LIN {X 0,Y 516.944,Z 452.093,A -85,B 0,C 180,E1 -4929.732,E2 -4929.732} C_VEL
LIN {X 0,Y 516.912,Z 452.096,A -85,B 0,C 180,E1 -4932.596,E2 -4932.596} C_VEL
LIN {X 0,Y 516.948,Z 452.092,A -85,B 0,C 180,E1 -4935.03,E2 -4935.03} C_VEL
LIN {X 0,Y 516.971,Z 452.089,A -85,B 0,C 180,E1 -4938.234,E2 -4938.234} C_VEL
LIN {X 0,Y 516.971,Z 452.089,A -85,B 0,C 180,E1 -4941.4,E2 -4941.4} C_VEL
LIN {X 0,Y 517.028,Z 452.081,A -85,B 0,C 180,E1 -4944.54,E2 -4944.54} C_VEL
LIN {X 0,Y 517.089,Z 452.074,A -85,B 0,C 180,E1 -4947.663,E2 -4947.663} C_VEL
LIN {X 0,Y 517.097,Z 452.071,A -85,B 0,C 180,E1 -4950.779,E2 -4950.779} C_VEL
LIN {X 0,Y 517.016,Z 452.085,A -85,B 0,C 180,E1 -4953.117,E2 -4953.117} C_VEL
LIN {X 0,Y 517.016,Z 452.085,A -85,B 0,C 180,E1 -4956.243,E2 -4956.243} C_VEL
LIN {X 0,Y 516.954,Z 452.092,A -85,B 0,C 180,E1 -4959.389,E2 -4959.389} C_VEL
LIN {X 0,Y 516.958,Z 452.09,A -85,B 0,C 180,E1 -4961.807,E2 -4961.807} C_VEL
LIN {X 0,Y 516.95,Z 452.09,A -85,B 0,C 180,E1 -4965.147,E2 -4965.147} C_VEL
LIN {X 0,Y 516.93,Z 452.093,A -85,B 0,C 180,E1 -4968.222,E2 -4968.222} C_VEL
LIN {X 0,Y 516.918,Z 452.097,A -85,B 0,C 180,E1 -4970.701,E2 -4970.701} C_VEL
LIN {X 0,Y 516.909,Z 452.097,A -85,B 0,C 180,E1 -4974.072,E2 -4974.072} C_VEL
LIN {X 0,Y 516.93,Z 452.097,A -85,B 0,C 180,E1 -4976.658,E2 -4976.658} C_VEL
LIN {X 0,Y 516.916,Z 452.096,A -85,B 0,C 180,E1 -4979.524,E2 -4979.524} C_VEL
LIN {X 0,Y 516.9,Z 452.098,A -85,B 0,C 180,E1 -4982.543,E2 -4982.543} C_VEL
LIN {X 0,Y 516.871,Z 452.1,A -85,B 0,C 180,E1 -4985.33,E2 -4985.33} C_VEL
LIN {X 0,Y 516.885,Z 452.101,A -85,B 0,C 180,E1 -4987.943,E2 -4987.943} C_VEL
LIN {X 0,Y 516.889,Z 452.101,A -85,B 0,C 180,E1 -4990.741,E2 -4990.741} C_VEL
LIN {X 0,Y 516.887,Z 452.099,A -85,B 0,C 180,E1 -4992.831,E2 -4992.831} C_VEL
LIN {X 0,Y 516.887,Z 452.099,A -85,B 0,C 180,E1 -4996.097,E2 -4996.097} C_VEL
LIN {X 0,Y 516.92,Z 452.098,A -85,B 0,C 180,E1 -4998.398,E2 -4998.398} C_VEL
LIN {X 0,Y 516.884,Z 452.099,A -85,B 0,C 180,E1 -5001.284,E2 -5001.284} C_VEL
LIN {X 0,Y 516.808,Z 452.109,A -85,B 0,C 180,E1 -5004.214,E2 -5004.214} C_VEL
LIN {X 0,Y 516.707,Z 452.125,A -85,B 0,C 180,E1 -5006.105,E2 -5006.105} C_VEL
LIN {X 0,Y 516.479,Z 452.226,A -85,B 0,C 180,E1 -5007.947,E2 -5007.947} C_VEL
LIN {X 0,Y 516.445,Z 455.171,A -85,B 0,C 180,E1 -5010.665,E2 -5010.665} C_VEL
LIN {X 0,Y 516.432,Z 458.051,A -85,B 0,C 180,E1 -5013.314,E2 -5013.314} C_VEL
LIN {X 0,Y 516.375,Z 460.913,A -85,B 0,C 180,E1 -5015.901,E2 -5015.901} C_VEL
LIN {X 0,Y 516.337,Z 463.731,A -85,B 0,C 180,E1 -5018.438,E2 -5018.438} C_VEL
LIN {X 0,Y 516.302,Z 466.547,A -85,B 0,C 180,E1 -5020.932,E2 -5020.932} C_VEL
LIN {X 0,Y 516.277,Z 469.313,A -85,B 0,C 180,E1 -5023.389,E2 -5023.389} C_VEL
LIN {X 0,Y 516.308,Z 472.56,A -85,B 0,C 180,E1 -5026.219,E2 -5026.219} C_VEL
LIN {X 0,Y 518.389,Z 484.619,A -85,B 0,C 180,E1 -5026.6,E2 -5026.6} C_VEL
LIN {X 0,Y 518.151,Z 497.874,A -85,B 0,C 180,E1 -5027.117,E2 -5027.117} C_VEL
LIN {X 0,Y 517.878,Z 509.167,A -85,B 0,C 180,E1 -5027.715,E2 -5027.715} C_VEL
LIN {X 0,Y 517.621,Z 519.986,A -85,B 0,C 180,E1 -5028.447,E2 -5028.447} C_VEL
LIN {X 0,Y 517.303,Z 530.501,A -85,B 0,C 180,E1 -5029.332,E2 -5029.332} C_VEL
LIN {X 0,Y 517.054,Z 539.091,A -85,B 0,C 180,E1 -5030.218,E2 -5030.218} C_VEL
LIN {X 0,Y 516.835,Z 546.997,A -85,B 0,C 180,E1 -5031.2,E2 -5031.2} C_VEL
LIN {X 0,Y 516.602,Z 554.73,A -85,B 0,C 180,E1 -5032.378,E2 -5032.378} C_VEL
LIN {X 0,Y 516.448,Z 561.797,A -85,B 0,C 180,E1 -5033.75,E2 -5033.75} C_VEL
LIN {X 0,Y 516.314,Z 566.51,A -85,B 0,C 180,E1 -5034.924,E2 -5034.924} C_VEL
LIN {X 0,Y 516.373,Z 570.109,A -85,B 0,C 180,E1 -5036.098,E2 -5036.098} C_VEL
LIN {X 0,Y 516.283,Z 571.978,A -85,B 0,C 180,E1 -5036.879,E2 -5036.879} C_VEL
LIN {X 0,Y 516.261,Z 573.384,A -85,B 0,C 180,E1 -5037.659,E2 -5037.659} C_VEL
LIN {X 0,Y 516.161,Z 575.003,A -85,B 0,C 180,E1 -5039.22,E2 -5039.22} C_VEL
LIN {X 0,Y 516.154,Z 575.245,A -85,B 0,C 180,E1 -5040,E2 -5040} C_VEL
LIN {X 0,Y 516.16,Z 575.064,A -85,B 0,C 180,E1 -5040.78,E2 -5040.78} C_VEL
LIN {X 0,Y 516.261,Z 573.525,A -85,B 0,C 180,E1 -5042.34,E2 -5042.34} C_VEL
LIN {X 0,Y 516.283,Z 572.181,A -85,B 0,C 180,E1 -5043.121,E2 -5043.121} C_VEL
LIN {X 0,Y 516.361,Z 569.332,A -85,B 0,C 180,E1 -5044.293,E2 -5044.293} C_VEL
LIN {X 0,Y 516.401,Z 565.469,A -85,B 0,C 180,E1 -5045.467,E2 -5045.467} C_VEL
LIN {X 0,Y 516.49,Z 559.63,A -85,B 0,C 180,E1 -5046.814,E2 -5046.814} C_VEL
LIN {X 0,Y 516.653,Z 552.961,A -85,B 0,C 180,E1 -5048.015,E2 -5048.015} C_VEL
LIN {X 0,Y 516.849,Z 544.818,A -85,B 0,C 180,E1 -5049.194,E2 -5049.194} C_VEL
LIN {X 0,Y 517.107,Z 536.463,A -85,B 0,C 180,E1 -5050.177,E2 -5050.177} C_VEL
LIN {X 0,Y 517.465,Z 526.118,A -85,B 0,C 180,E1 -5051.159,E2 -5051.159} C_VEL
LIN {X 0,Y 517.787,Z 514.576,A -85,B 0,C 180,E1 -5052.037,E2 -5052.037} C_VEL
LIN {X 0,Y 518.071,Z 502.798,A -85,B 0,C 180,E1 -5052.735,E2 -5052.735} C_VEL
LIN {X 0,Y 518.336,Z 490.688,A -85,B 0,C 180,E1 -5053.277,E2 -5053.277} C_VEL
LIN {X 0,Y 518.251,Z 483.303,A -85,B 0,C 180,E1 -5053.541,E2 -5053.541} C_VEL
LIN {X 0,Y 516.316,Z 472.997,A -85,B 0,C 180,E1 -5053.881,E2 -5053.881} C_VEL
LIN {X 0,Y 516.34,Z 470.114,A -85,B 0,C 180,E1 -5056.609,E2 -5056.609} C_VEL
LIN {X 0,Y 516.386,Z 467.623,A -85,B 0,C 180,E1 -5059.065,E2 -5059.065} C_VEL
LIN {X 0,Y 516.433,Z 465.115,A -85,B 0,C 180,E1 -5061.558,E2 -5061.558} C_VEL
LIN {X 0,Y 516.557,Z 462.467,A -85,B 0,C 180,E1 -5064.277,E2 -5064.277} C_VEL
LIN {X 0,Y 516.677,Z 459.367,A -85,B 0,C 180,E1 -5067.547,E2 -5067.547} C_VEL
LIN {X 0,Y 516.708,Z 456.952,A -85,B 0,C 180,E1 -5070.216,E2 -5070.216} C_VEL
LIN {X 0,Y 516.837,Z 454.601,A -85,B 0,C 180,E1 -5072.951,E2 -5072.951} C_VEL
LIN {X 0,Y 516.847,Z 452.379,A -85,B 0,C 180,E1 -5075.782,E2 -5075.782} C_VEL
LIN {X 0,Y 516.883,Z 452.104,A -85,B 0,C 180,E1 -5077.943,E2 -5077.943} C_VEL
LIN {X 0,Y 516.887,Z 452.102,A -85,B 0,C 180,E1 -5080.741,E2 -5080.741} C_VEL
LIN {X 0,Y 516.908,Z 452.1,A -85,B 0,C 180,E1 -5082.829,E2 -5082.829} C_VEL
LIN {X 0,Y 516.926,Z 452.098,A -85,B 0,C 180,E1 -5085.01,E2 -5085.01} C_VEL
LIN {X 0,Y 516.918,Z 452.098,A -85,B 0,C 180,E1 -5088.398,E2 -5088.398} C_VEL
LIN {X 0,Y 516.932,Z 452.198,A -85,B 0,C 180,E1 -5089.263,E2 -5089.263} C_VEL
LIN {X 0,Y 517.422,Z 454.988,A -85,B 0,C 180,E1 -5091.332,E2 -5091.332} C_VEL
LIN {X 0,Y 518.009,Z 458.473,A -85,B 0,C 180,E1 -5093.347,E2 -5093.347} C_VEL
LIN {X 0,Y 518.115,Z 462.532,A -85,B 0,C 180,E1 -5095.27,E2 -5095.27} C_VEL
LIN {X 0,Y 517.661,Z 469.386,A -85,B 0,C 180,E1 -5098.029,E2 -5098.029} C_VEL
LIN {X 0,Y 517.314,Z 476.785,A -85,B 0,C 180,E1 -5100.72,E2 -5100.72} C_VEL
LIN {X 0,Y 517.151,Z 484.588,A -85,B 0,C 180,E1 -5103.355,E2 -5103.355} C_VEL
LIN {X 0,Y 517.002,Z 492.652,A -85,B 0,C 180,E1 -5105.932,E2 -5105.932} C_VEL
LIN {X 0,Y 516.828,Z 502.252,A -85,B 0,C 180,E1 -5108.878,E2 -5108.878} C_VEL
LIN {X 0,Y 516.716,Z 511.979,A -85,B 0,C 180,E1 -5111.77,E2 -5111.77} C_VEL
LIN {X 0,Y 516.633,Z 523.068,A -85,B 0,C 180,E1 -5115.021,E2 -5115.021} C_VEL
LIN {X 0,Y 516.569,Z 526.747,A -85,B 0,C 180,E1 -5116.101,E2 -5116.101} C_VEL
LIN {X 0,Y 518.446,Z 539.825,A -85,B 0,C 180,E1 -5116.452,E2 -5116.452} C_VEL
LIN {X 0,Y 518.221,Z 551.89,A -85,B 0,C 180,E1 -5116.87,E2 -5116.87} C_VEL
LIN {X 0,Y 517.963,Z 564.239,A -85,B 0,C 180,E1 -5117.461,E2 -5117.461} C_VEL
LIN {X 0,Y 517.647,Z 575.446,A -85,B 0,C 180,E1 -5118.154,E2 -5118.154} C_VEL
LIN {X 0,Y 517.345,Z 586.795,A -85,B 0,C 180,E1 -5119.036,E2 -5119.036} C_VEL
LIN {X 0,Y 517.018,Z 596.875,A -85,B 0,C 180,E1 -5120.019,E2 -5120.019} C_VEL
LIN {X 0,Y 516.77,Z 606.653,A -85,B 0,C 180,E1 -5121.199,E2 -5121.199} C_VEL
LIN {X 0,Y 516.563,Z 614.431,A -85,B 0,C 180,E1 -5122.377,E2 -5122.377} C_VEL
LIN {X 0,Y 516.427,Z 621.594,A -85,B 0,C 180,E1 -5123.75,E2 -5123.75} C_VEL
LIN {X 0,Y 516.314,Z 626.349,A -85,B 0,C 180,E1 -5124.924,E2 -5124.924} C_VEL
LIN {X 0,Y 516.354,Z 629.957,A -85,B 0,C 180,E1 -5126.098,E2 -5126.098} C_VEL
LIN {X 0,Y 516.282,Z 631.806,A -85,B 0,C 180,E1 -5126.879,E2 -5126.879} C_VEL
LIN {X 0,Y 516.261,Z 633.192,A -85,B 0,C 180,E1 -5127.659,E2 -5127.659} C_VEL
LIN {X 0,Y 516.16,Z 634.785,A -85,B 0,C 180,E1 -5129.22,E2 -5129.22} C_VEL
LIN {X 0,Y 516.154,Z 635,A -85,B 0,C 180,E1 -5130,E2 -5130} C_VEL
LIN {X 0,Y 516.192,Z 634.183,A -85,B 0,C 180,E1 -5131.56,E2 -5131.56} C_VEL
LIN {X 0,Y 516.26,Z 633.195,A -85,B 0,C 180,E1 -5132.341,E2 -5132.341} C_VEL
LIN {X 0,Y 516.282,Z 631.81,A -85,B 0,C 180,E1 -5133.121,E2 -5133.121} C_VEL
LIN {X 0,Y 516.343,Z 628.891,A -85,B 0,C 180,E1 -5134.293,E2 -5134.293} C_VEL
LIN {X 0,Y 516.405,Z 624.912,A -85,B 0,C 180,E1 -5135.467,E2 -5135.467} C_VEL
LIN {X 0,Y 516.479,Z 618.972,A -85,B 0,C 180,E1 -5136.798,E2 -5136.798} C_VEL
LIN {X 0,Y 516.641,Z 612.041,A -85,B 0,C 180,E1 -5138.015,E2 -5138.015} C_VEL
LIN {X 0,Y 516.844,Z 603.701,A -85,B 0,C 180,E1 -5139.194,E2 -5139.194} C_VEL
LIN {X 0,Y 517.058,Z 595.147,A -85,B 0,C 180,E1 -5140.178,E2 -5140.178} C_VEL
LIN {X 0,Y 517.416,Z 584.586,A -85,B 0,C 180,E1 -5141.16,E2 -5141.16} C_VEL
LIN {X 0,Y 517.752,Z 572.753,A -85,B 0,C 180,E1 -5142.043,E2 -5142.043} C_VEL
LIN {X 0,Y 518.042,Z 560.744,A -85,B 0,C 180,E1 -5142.736,E2 -5142.736} C_VEL
LIN {X 0,Y 518.322,Z 548.322,A -85,B 0,C 180,E1 -5143.277,E2 -5143.277} C_VEL
LIN {X 0,Y 518.25,Z 537.856,A -85,B 0,C 180,E1 -5143.616,E2 -5143.616} C_VEL
LIN {X 0,Y 516.585,Z 527.009,A -85,B 0,C 180,E1 -5143.924,E2 -5143.924} C_VEL
LIN {X 0,Y 516.709,Z 516.721,A -85,B 0,C 180,E1 -5147.004,E2 -5147.004} C_VEL
LIN {X 0,Y 516.841,Z 507.225,A -85,B 0,C 180,E1 -5149.874,E2 -5149.874} C_VEL
LIN {X 0,Y 516.998,Z 497.939,A -85,B 0,C 180,E1 -5152.794,E2 -5152.794} C_VEL
LIN {X 0,Y 517.231,Z 488.663,A -85,B 0,C 180,E1 -5155.773,E2 -5155.773} C_VEL
LIN {X 0,Y 517.463,Z 480.76,A -85,B 0,C 180,E1 -5158.383,E2 -5158.383} C_VEL
LIN {X 0,Y 517.775,Z 472.402,A -85,B 0,C 180,E1 -5161.226,E2 -5161.226} C_VEL
LIN {X 0,Y 518.065,Z 464.125,A -85,B 0,C 180,E1 -5164.155,E2 -5164.155} C_VEL
LIN {X 0,Y 518.147,Z 459.971,A -85,B 0,C 180,E1 -5165.679,E2 -5165.679} C_VEL
LIN {X 0,Y 517.232,Z 454.031,A -85,B 0,C 180,E1 -5167.993,E2 -5167.993} C_VEL
LIN {X 0,Y 516.886,Z 452.102,A -85,B 0,C 180,E1 -5168.835,E2 -5168.835} C_VEL
LIN {X 0,Y 516.915,Z 452.098,A -85,B 0,C 180,E1 -5171.775,E2 -5171.775} C_VEL
LIN {X 0,Y 516.925,Z 452.095,A -85,B 0,C 180,E1 -5175.01,E2 -5175.01} C_VEL
LIN {X 0,Y 516.918,Z 452.095,A -85,B 0,C 180,E1 -5178.398,E2 -5178.398} C_VEL
LIN {X 0,Y 516.881,Z 452.099,A -85,B 0,C 180,E1 -5181.284,E2 -5181.284} C_VEL
LIN {X 0,Y 516.873,Z 452.103,A -85,B 0,C 180,E1 -5184.22,E2 -5184.22} C_VEL
LIN {X 0,Y 516.896,Z 452.101,A -85,B 0,C 180,E1 -5187.053,E2 -5187.053} C_VEL
LIN {X 0,Y 516.894,Z 452.099,A -85,B 0,C 180,E1 -5189.796,E2 -5189.796} C_VEL
LIN {X 0,Y 516.93,Z 452.093,A -85,B 0,C 180,E1 -5192.467,E2 -5192.467} C_VEL
LIN {X 0,Y 516.906,Z 452.097,A -85,B 0,C 180,E1 -5195.072,E2 -5195.072} C_VEL
LIN {X 0,Y 516.888,Z 452.099,A -85,B 0,C 180,E1 -5198.462,E2 -5198.462} C_VEL
LIN {X 0,Y 516.906,Z 452.101,A -85,B 0,C 180,E1 -5200.955,E2 -5200.955} C_VEL
LIN {X 0,Y 516.916,Z 452.094,A -85,B 0,C 180,E1 -5203.41,E2 -5203.41} C_VEL
LIN {X 0,Y 516.898,Z 452.101,A -85,B 0,C 180,E1 -5205.834,E2 -5205.834} C_VEL
LIN {X 0,Y 516.968,Z 452.089,A -85,B 0,C 180,E1 -5208.234,E2 -5208.234} C_VEL
LIN {X 0,Y 516.97,Z 452.088,A -85,B 0,C 180,E1 -5211.4,E2 -5211.4} C_VEL
LIN {X 0,Y 517.012,Z 452.086,A -85,B 0,C 180,E1 -5213.757,E2 -5213.757} C_VEL
LIN {X 0,Y 517.085,Z 452.073,A -85,B 0,C 180,E1 -5217.663,E2 -5217.663} C_VEL
LIN {X 0,Y 517.098,Z 452.073,A -85,B 0,C 180,E1 -5220.779,E2 -5220.779} C_VEL
LIN {X 0,Y 517.015,Z 452.084,A -85,B 0,C 180,E1 -5223.117,E2 -5223.117} C_VEL
LIN {X 0,Y 517.013,Z 452.086,A -85,B 0,C 180,E1 -5226.243,E2 -5226.243} C_VEL
LIN {X 0,Y 516.956,Z 452.092,A -85,B 0,C 180,E1 -5229.389,E2 -5229.389} C_VEL
LIN {X 0,Y 516.955,Z 452.09,A -85,B 0,C 180,E1 -5231.807,E2 -5231.807} C_VEL
LIN {X 0,Y 516.948,Z 452.094,A -85,B 0,C 180,E1 -5235.147,E2 -5235.147} C_VEL
LIN {X 0,Y 516.928,Z 452.095,A -85,B 0,C 180,E1 -5238.222,E2 -5238.222} C_VEL
LIN {X 0,Y 516.916,Z 452.095,A -85,B 0,C 180,E1 -5240.702,E2 -5240.702} C_VEL
LIN {X 0,Y 516.906,Z 452.096,A -85,B 0,C 180,E1 -5244.073,E2 -5244.073} C_VEL
LIN {X 0,Y 516.929,Z 452.094,A -85,B 0,C 180,E1 -5246.658,E2 -5246.658} C_VEL
LIN {X 0,Y 516.914,Z 452.098,A -85,B 0,C 180,E1 -5249.524,E2 -5249.524} C_VEL
LIN {X 0,Y 516.901,Z 452.101,A -85,B 0,C 180,E1 -5252.544,E2 -5252.544} C_VEL
LIN {X 0,Y 516.884,Z 452.101,A -85,B 0,C 180,E1 -5255.332,E2 -5255.332} C_VEL
LIN {X 0,Y 516.884,Z 452.099,A -85,B 0,C 180,E1 -5257.943,E2 -5257.943} C_VEL
LIN {X 0,Y 516.887,Z 452.099,A -85,B 0,C 180,E1 -5260.742,E2 -5260.742} C_VEL
LIN {X 0,Y 516.908,Z 452.096,A -85,B 0,C 180,E1 -5262.829,E2 -5262.829} C_VEL
LIN {X 0,Y 516.926,Z 452.097,A -85,B 0,C 180,E1 -5265.01,E2 -5265.01} C_VEL
LIN {X 0,Y 516.917,Z 452.097,A -85,B 0,C 180,E1 -5268.399,E2 -5268.399} C_VEL
LIN {X 0,Y 516.885,Z 452.099,A -85,B 0,C 180,E1 -5270.301,E2 -5270.301} C_VEL
LIN {X 0,Y 516.214,Z 452.185,A -85,B 0,C 180,E1 -5270.951,E2 -5270.951} C_VEL
LIN {X 0,Y 513.369,Z 452.537,A -85,B 0,C 180,E1 -5272.007,E2 -5272.007} C_VEL
LIN {X 0,Y 510.962,Z 452.839,A -85,B 0,C 180,E1 -5272.857,E2 -5272.857} C_VEL
LIN {X 0,Y 509.922,Z 452.966,A -85,B 0,C 180,E1 -5273.514,E2 -5273.514} C_VEL
LIN {X 0,Y 509.833,Z 452.977,A -85,B 0,C 180,E1 -5273.736,E2 -5273.736} C_VEL
LIN {X 0,Y 509.865,Z 452.973,A -85,B 0,C 180,E1 -5276.54,E2 -5276.54} C_VEL
LIN {X 0,Y 509.85,Z 452.978,A -85,B 0,C 180,E1 -5279.334,E2 -5279.334} C_VEL
LIN {X 0,Y 509.895,Z 452.973,A -85,B 0,C 180,E1 -5282.055,E2 -5282.055} C_VEL
LIN {X 0,Y 509.881,Z 452.972,A -85,B 0,C 180,E1 -5284.704,E2 -5284.704} C_VEL
LIN {X 0,Y 509.831,Z 452.978,A -85,B 0,C 180,E1 -5287.458,E2 -5287.458} C_VEL
LIN {X 0,Y 509.921,Z 452.969,A -85,B 0,C 180,E1 -5289.845,E2 -5289.845} C_VEL
LIN {X 0,Y 509.879,Z 452.974,A -85,B 0,C 180,E1 -5293.175,E2 -5293.175} C_VEL
LIN {X 0,Y 509.869,Z 452.973,A -85,B 0,C 180,E1 -5295.634,E2 -5295.634} C_VEL
LIN {X 0,Y 509.919,Z 452.967,A -85,B 0,C 180,E1 -5298.875,E2 -5298.875} C_VEL
LIN {X 0,Y 509.957,Z 452.964,A -85,B 0,C 180,E1 -5302.079,E2 -5302.079} C_VEL
LIN {X 0,Y 509.978,Z 452.959,A -85,B 0,C 180,E1 -5304.464,E2 -5304.464} C_VEL
LIN {X 0,Y 510.06,Z 452.95,A -85,B 0,C 180,E1 -5307.631,E2 -5307.631} C_VEL
LIN {X 0,Y 510.068,Z 452.947,A -85,B 0,C 180,E1 -5310.79,E2 -5310.79} C_VEL
LIN {X 0,Y 509.958,Z 452.964,A -85,B 0,C 180,E1 -5313.16,E2 -5313.16} C_VEL
LIN {X 0,Y 509.984,Z 452.962,A -85,B 0,C 180,E1 -5316.33,E2 -5316.33} C_VEL
LIN {X 0,Y 509.895,Z 452.972,A -85,B 0,C 180,E1 -5319.521,E2 -5319.521} C_VEL
LIN {X 0,Y 509.91,Z 452.968,A -85,B 0,C 180,E1 -5321.932,E2 -5321.932} C_VEL
LIN {X 0,Y 509.9,Z 452.968,A -85,B 0,C 180,E1 -5325.242,E2 -5325.242} C_VEL
LIN {X 0,Y 509.887,Z 452.971,A -85,B 0,C 180,E1 -5327.998,E2 -5327.998} C_VEL
LIN {X 0,Y 509.856,Z 452.975,A -85,B 0,C 180,E1 -5331.002,E2 -5331.002} C_VEL
LIN {X 0,Y 509.87,Z 452.972,A -85,B 0,C 180,E1 -5334.426,E2 -5334.426} C_VEL
LIN {X 0,Y 509.889,Z 452.973,A -85,B 0,C 180,E1 -5337.056,E2 -5337.056} C_VEL
LIN {X 0,Y 509.862,Z 452.977,A -85,B 0,C 180,E1 -5339.751,E2 -5339.751} C_VEL
LIN {X 0,Y 509.878,Z 452.974,A -85,B 0,C 180,E1 -5342.774,E2 -5342.774} C_VEL
LIN {X 0,Y 509.831,Z 452.978,A -85,B 0,C 180,E1 -5345.578,E2 -5345.578} C_VEL
LIN {X 0,Y 509.855,Z 452.974,A -85,B 0,C 180,E1 -5348.338,E2 -5348.338} C_VEL
LIN {X 0,Y 509.861,Z 452.974,A -85,B 0,C 180,E1 -5351.425,E2 -5351.425} C_VEL
LIN {X 0,Y 509.843,Z 452.974,A -85,B 0,C 180,E1 -5354.67,E2 -5354.67} C_VEL
LIN {X 0,Y 509.862,Z 452.975,A -85,B 0,C 180,E1 -5358.103,E2 -5358.103} C_VEL
LIN {X 0,Y 509.85,Z 452.975,A -85,B 0,C 180,E1 -5360.647,E2 -5360.647} C_VEL
LIN {X 0,Y 509.79,Z 452.984,A -85,B 0,C 180,E1 -5363.644,E2 -5363.644} C_VEL
LIN {X 0,Y 509.692,Z 452.999,A -85,B 0,C 180,E1 -5365.825,E2 -5365.825} C_VEL
LIN {X 0,Y 509.487,Z 453.025,A -85,B 0,C 180,E1 -5367.454,E2 -5367.454} C_VEL
LIN {X 0,Y 509.405,Z 453.343,A -85,B 0,C 180,E1 -5368.381,E2 -5368.381} C_VEL
LIN {X 0,Y 509.361,Z 456.296,A -85,B 0,C 180,E1 -5371.123,E2 -5371.123} C_VEL
LIN {X 0,Y 509.394,Z 459.196,A -85,B 0,C 180,E1 -5373.8,E2 -5373.8} C_VEL
LIN {X 0,Y 509.272,Z 462.075,A -85,B 0,C 180,E1 -5376.409,E2 -5376.409} C_VEL
LIN {X 0,Y 509.248,Z 464.917,A -85,B 0,C 180,E1 -5378.972,E2 -5378.972} C_VEL
LIN {X 0,Y 509.246,Z 467.715,A -85,B 0,C 180,E1 -5381.493,E2 -5381.493} C_VEL
LIN {X 0,Y 509.202,Z 470.534,A -85,B 0,C 180,E1 -5383.976,E2 -5383.976} C_VEL
LIN {X 0,Y 509.235,Z 472.857,A -85,B 0,C 180,E1 -5386.024,E2 -5386.024} C_VEL
LIN {X 0,Y 511.498,Z 485.521,A -85,B 0,C 180,E1 -5386.441,E2 -5386.441} C_VEL
LIN {X 0,Y 511.248,Z 498.027,A -85,B 0,C 180,E1 -5386.94,E2 -5386.94} C_VEL
LIN {X 0,Y 510.931,Z 510.045,A -85,B 0,C 180,E1 -5387.589,E2 -5387.589} C_VEL
LIN {X 0,Y 510.611,Z 521.491,A -85,B 0,C 180,E1 -5388.387,E2 -5388.387} C_VEL
LIN {X 0,Y 510.32,Z 531.808,A -85,B 0,C 180,E1 -5389.285,E2 -5389.285} C_VEL
LIN {X 0,Y 510.007,Z 541.084,A -85,B 0,C 180,E1 -5390.281,E2 -5390.281} C_VEL
LIN {X 0,Y 509.721,Z 550.047,A -85,B 0,C 180,E1 -5391.476,E2 -5391.476} C_VEL
LIN {X 0,Y 509.496,Z 557.271,A -85,B 0,C 180,E1 -5392.669,E2 -5392.669} C_VEL
LIN {X 0,Y 509.388,Z 562.137,A -85,B 0,C 180,E1 -5393.663,E2 -5393.663} C_VEL
LIN {X 0,Y 509.248,Z 566.868,A -85,B 0,C 180,E1 -5394.853,E2 -5394.853} C_VEL
LIN {X 0,Y 509.303,Z 570.484,A -85,B 0,C 180,E1 -5396.044,E2 -5396.044} C_VEL
LIN {X 0,Y 509.202,Z 572.366,A -85,B 0,C 180,E1 -5396.835,E2 -5396.835} C_VEL
LIN {X 0,Y 509.19,Z 573.779,A -85,B 0,C 180,E1 -5397.627,E2 -5397.627} C_VEL
LIN {X 0,Y 509.074,Z 575.409,A -85,B 0,C 180,E1 -5399.209,E2 -5399.209} C_VEL
LIN {X 0,Y 509.067,Z 575.657,A -85,B 0,C 180,E1 -5400,E2 -5400} C_VEL
LIN {X 0,Y 509.074,Z 575.479,A -85,B 0,C 180,E1 -5400.791,E2 -5400.791} C_VEL
LIN {X 0,Y 509.189,Z 573.94,A -85,B 0,C 180,E1 -5402.373,E2 -5402.373} C_VEL
LIN {X 0,Y 509.216,Z 572.595,A -85,B 0,C 180,E1 -5403.165,E2 -5403.165} C_VEL
LIN {X 0,Y 509.283,Z 569.742,A -85,B 0,C 180,E1 -5404.353,E2 -5404.353} C_VEL
LIN {X 0,Y 509.341,Z 565.869,A -85,B 0,C 180,E1 -5405.543,E2 -5405.543} C_VEL
LIN {X 0,Y 509.455,Z 560.213,A -85,B 0,C 180,E1 -5406.868,E2 -5406.868} C_VEL
LIN {X 0,Y 509.625,Z 553.326,A -85,B 0,C 180,E1 -5408.126,E2 -5408.126} C_VEL
LIN {X 0,Y 509.84,Z 545.162,A -85,B 0,C 180,E1 -5409.321,E2 -5409.321} C_VEL
LIN {X 0,Y 510.119,Z 536.779,A -85,B 0,C 180,E1 -5410.317,E2 -5410.317} C_VEL
LIN {X 0,Y 510.516,Z 526.397,A -85,B 0,C 180,E1 -5411.313,E2 -5411.313} C_VEL
LIN {X 0,Y 510.851,Z 514.832,A -85,B 0,C 180,E1 -5412.203,E2 -5412.203} C_VEL
LIN {X 0,Y 511.145,Z 502.988,A -85,B 0,C 180,E1 -5412.91,E2 -5412.91} C_VEL
LIN {X 0,Y 511.435,Z 490.856,A -85,B 0,C 180,E1 -5413.459,E2 -5413.459} C_VEL
LIN {X 0,Y 511.325,Z 484.198,A -85,B 0,C 180,E1 -5413.702,E2 -5413.702} C_VEL
LIN {X 0,Y 509.675,Z 475.381,A -85,B 0,C 180,E1 -5413.992,E2 -5413.992} C_VEL
LIN {X 0,Y 509.261,Z 473.536,A -85,B 0,C 180,E1 -5414.061,E2 -5414.061} C_VEL
LIN {X 0,Y 509.281,Z 470.642,A -85,B 0,C 180,E1 -5416.846,E2 -5416.846} C_VEL
LIN {X 0,Y 509.328,Z 468.116,A -85,B 0,C 180,E1 -5419.34,E2 -5419.34} C_VEL
LIN {X 0,Y 509.418,Z 465.081,A -85,B 0,C 180,E1 -5422.43,E2 -5422.43} C_VEL
LIN {X 0,Y 509.512,Z 462.323,A -85,B 0,C 180,E1 -5425.315,E2 -5425.315} C_VEL
LIN {X 0,Y 509.614,Z 459.818,A -85,B 0,C 180,E1 -5428.04,E2 -5428.04} C_VEL
LIN {X 0,Y 509.755,Z 457.024,A -85,B 0,C 180,E1 -5431.262,E2 -5431.262} C_VEL
LIN {X 0,Y 509.868,Z 454.499,A -85,B 0,C 180,E1 -5434.412,E2 -5434.412} C_VEL
LIN {X 0,Y 509.801,Z 453.126,A -85,B 0,C 180,E1 -5436.355,E2 -5436.355} C_VEL
LIN {X 0,Y 509.849,Z 452.979,A -85,B 0,C 180,E1 -5439.352,E2 -5439.352} C_VEL
LIN {X 0,Y 509.851,Z 452.98,A -85,B 0,C 180,E1 -5442.488,E2 -5442.488} C_VEL
LIN {X 0,Y 509.86,Z 452.978,A -85,B 0,C 180,E1 -5445.332,E2 -5445.332} C_VEL
LIN {X 0,Y 509.877,Z 453.077,A -85,B 0,C 180,E1 -5448.576,E2 -5448.576} C_VEL
LIN {X 0,Y 510.357,Z 455.629,A -85,B 0,C 180,E1 -5450.694,E2 -5450.694} C_VEL
LIN {X 0,Y 510.947,Z 459.187,A -85,B 0,C 180,E1 -5452.919,E2 -5452.919} C_VEL
LIN {X 0,Y 511.191,Z 462.758,A -85,B 0,C 180,E1 -5454.73,E2 -5454.73} C_VEL
LIN {X 0,Y 510.806,Z 468.16,A -85,B 0,C 180,E1 -5457.064,E2 -5457.064} C_VEL
LIN {X 0,Y 510.404,Z 476.322,A -85,B 0,C 180,E1 -5460.167,E2 -5460.167} C_VEL
LIN {X 0,Y 510.158,Z 484.319,A -85,B 0,C 180,E1 -5462.96,E2 -5462.96} C_VEL
LIN {X 0,Y 509.931,Z 493.641,A -85,B 0,C 180,E1 -5466.01,E2 -5466.01} C_VEL
LIN {X 0,Y 509.767,Z 503.185,A -85,B 0,C 180,E1 -5468.995,E2 -5468.995} C_VEL
LIN {X 0,Y 509.593,Z 513.479,A -85,B 0,C 180,E1 -5472.103,E2 -5472.103} C_VEL
LIN {X 0,Y 509.537,Z 524.091,A -85,B 0,C 180,E1 -5475.27,E2 -5475.27} C_VEL
LIN {X 0,Y 509.485,Z 526.45,A -85,B 0,C 180,E1 -5475.916,E2 -5475.916} C_VEL
LIN {X 0,Y 511.398,Z 539.42,A -85,B 0,C 180,E1 -5476.274,E2 -5476.274} C_VEL
LIN {X 0,Y 511.253,Z 552.277,A -85,B 0,C 180,E1 -5476.738,E2 -5476.738} C_VEL
LIN {X 0,Y 510.942,Z 564.881,A -85,B 0,C 180,E1 -5477.364,E2 -5477.364} C_VEL
LIN {X 0,Y 510.616,Z 576.136,A -85,B 0,C 180,E1 -5478.085,E2 -5478.085} C_VEL
LIN {X 0,Y 510.29,Z 587.242,A -85,B 0,C 180,E1 -5478.983,E2 -5478.983} C_VEL
LIN {X 0,Y 509.979,Z 596.274,A -85,B 0,C 180,E1 -5479.88,E2 -5479.88} C_VEL
LIN {X 0,Y 509.711,Z 606.09,A -85,B 0,C 180,E1 -5481.076,E2 -5481.076} C_VEL
LIN {X 0,Y 509.494,Z 613.907,A -85,B 0,C 180,E1 -5482.271,E2 -5482.271} C_VEL
LIN {X 0,Y 509.326,Z 621.095,A -85,B 0,C 180,E1 -5483.662,E2 -5483.662} C_VEL
LIN {X 0,Y 509.248,Z 625.882,A -85,B 0,C 180,E1 -5484.853,E2 -5484.853} C_VEL
LIN {X 0,Y 509.268,Z 629.542,A -85,B 0,C 180,E1 -5486.043,E2 -5486.043} C_VEL
LIN {X 0,Y 509.2,Z 631.427,A -85,B 0,C 180,E1 -5486.835,E2 -5486.835} C_VEL
LIN {X 0,Y 509.189,Z 632.839,A -85,B 0,C 180,E1 -5487.627,E2 -5487.627} C_VEL
LIN {X 0,Y 509.073,Z 634.457,A -85,B 0,C 180,E1 -5489.209,E2 -5489.209} C_VEL
LIN {X 0,Y 509.065,Z 634.679,A -85,B 0,C 180,E1 -5490,E2 -5490} C_VEL
LIN {X 0,Y 509.112,Z 633.856,A -85,B 0,C 180,E1 -5491.582,E2 -5491.582} C_VEL
LIN {X 0,Y 509.189,Z 632.859,A -85,B 0,C 180,E1 -5492.373,E2 -5492.373} C_VEL
LIN {X 0,Y 509.2,Z 631.453,A -85,B 0,C 180,E1 -5493.165,E2 -5493.165} C_VEL
LIN {X 0,Y 509.231,Z 628.497,A -85,B 0,C 180,E1 -5494.353,E2 -5494.353} C_VEL
LIN {X 0,Y 509.322,Z 624.494,A -85,B 0,C 180,E1 -5495.543,E2 -5495.543} C_VEL
LIN {X 0,Y 509.402,Z 618.785,A -85,B 0,C 180,E1 -5496.844,E2 -5496.844} C_VEL
LIN {X 0,Y 509.572,Z 611.594,A -85,B 0,C 180,E1 -5498.127,E2 -5498.127} C_VEL
LIN {X 0,Y 509.781,Z 603.24,A -85,B 0,C 180,E1 -5499.322,E2 -5499.322} C_VEL
LIN {X 0,Y 510.031,Z 594.666,A -85,B 0,C 180,E1 -5500.319,E2 -5500.319} C_VEL
LIN {X 0,Y 510.405,Z 584.084,A -85,B 0,C 180,E1 -5501.316,E2 -5501.316} C_VEL
LIN {X 0,Y 510.742,Z 572.234,A -85,B 0,C 180,E1 -5502.211,E2 -5502.211} C_VEL
LIN {X 0,Y 511.065,Z 560.194,A -85,B 0,C 180,E1 -5502.913,E2 -5502.913} C_VEL
LIN {X 0,Y 511.397,Z 547.768,A -85,B 0,C 180,E1 -5503.46,E2 -5503.46} C_VEL
LIN {X 0,Y 511.381,Z 539.106,A -85,B 0,C 180,E1 -5503.752,E2 -5503.752} C_VEL
LIN {X 0,Y 509.491,Z 526.74,A -85,B 0,C 180,E1 -5504.096,E2 -5504.096} C_VEL
LIN {X 0,Y 509.601,Z 517.781,A -85,B 0,C 180,E1 -5506.835,E2 -5506.835} C_VEL
LIN {X 0,Y 509.784,Z 508.375,A -85,B 0,C 180,E1 -5509.741,E2 -5509.741} C_VEL
LIN {X 0,Y 509.945,Z 499.057,A -85,B 0,C 180,E1 -5512.699,E2 -5512.699} C_VEL
LIN {X 0,Y 510.213,Z 489.828,A -85,B 0,C 180,E1 -5515.715,E2 -5515.715} C_VEL
LIN {X 0,Y 510.444,Z 482.367,A -85,B 0,C 180,E1 -5518.215,E2 -5518.215} C_VEL
LIN {X 0,Y 510.744,Z 474.201,A -85,B 0,C 180,E1 -5521.032,E2 -5521.032} C_VEL
LIN {X 0,Y 511.062,Z 466.34,A -85,B 0,C 180,E1 -5523.845,E2 -5523.845} C_VEL
LIN {X 0,Y 511.174,Z 461.088,A -85,B 0,C 180,E1 -5525.789,E2 -5525.789} C_VEL
LIN {X 0,Y 510.134,Z 454.722,A -85,B 0,C 180,E1 -5528.313,E2 -5528.313} C_VEL
LIN {X 0,Y 509.846,Z 452.98,A -85,B 0,C 180,E1 -5529.098,E2 -5529.098} C_VEL
LIN {X 0,Y 509.859,Z 452.976,A -85,B 0,C 180,E1 -5531.897,E2 -5531.897} C_VEL
LIN {X 0,Y 509.859,Z 452.974,A -85,B 0,C 180,E1 -5535.332,E2 -5535.332} C_VEL
LIN {X 0,Y 509.859,Z 452.974,A -85,B 0,C 180,E1 -5538.575,E2 -5538.575} C_VEL
LIN {X 0,Y 509.852,Z 452.974,A -85,B 0,C 180,E1 -5541.787,E2 -5541.787} C_VEL
LIN {X 0,Y 509.832,Z 452.978,A -85,B 0,C 180,E1 -5544.622,E2 -5544.622} C_VEL
LIN {X 0,Y 509.863,Z 452.973,A -85,B 0,C 180,E1 -5547.481,E2 -5547.481} C_VEL
LIN {X 0,Y 509.86,Z 452.978,A -85,B 0,C 180,E1 -5550.274,E2 -5550.274} C_VEL
LIN {X 0,Y 509.887,Z 452.973,A -85,B 0,C 180,E1 -5552.944,E2 -5552.944} C_VEL
LIN {X 0,Y 509.858,Z 452.973,A -85,B 0,C 180,E1 -5555.573,E2 -5555.573} C_VEL
LIN {X 0,Y 509.853,Z 452.976,A -85,B 0,C 180,E1 -5558.998,E2 -5558.998} C_VEL
LIN {X 0,Y 509.891,Z 452.969,A -85,B 0,C 180,E1 -5561.999,E2 -5561.999} C_VEL
LIN {X 0,Y 509.913,Z 452.968,A -85,B 0,C 180,E1 -5564.819,E2 -5564.819} C_VEL
LIN {X 0,Y 509.903,Z 452.968,A -85,B 0,C 180,E1 -5568.124,E2 -5568.124} C_VEL
LIN {X 0,Y 509.917,Z 452.966,A -85,B 0,C 180,E1 -5571.28,E2 -5571.28} C_VEL
LIN {X 0,Y 509.981,Z 452.962,A -85,B 0,C 180,E1 -5573.671,E2 -5573.671} C_VEL
LIN {X 0,Y 510.056,Z 452.948,A -85,B 0,C 180,E1 -5577.631,E2 -5577.631} C_VEL
LIN {X 0,Y 510.068,Z 452.949,A -85,B 0,C 180,E1 -5580.79,E2 -5580.79} C_VEL
LIN {X 0,Y 509.957,Z 452.963,A -85,B 0,C 180,E1 -5583.16,E2 -5583.16} C_VEL
LIN {X 0,Y 509.981,Z 452.961,A -85,B 0,C 180,E1 -5586.33,E2 -5586.33} C_VEL
LIN {X 0,Y 509.919,Z 452.968,A -85,B 0,C 180,E1 -5588.72,E2 -5588.72} C_VEL
LIN {X 0,Y 509.907,Z 452.968,A -85,B 0,C 180,E1 -5591.932,E2 -5591.932} C_VEL
LIN {X 0,Y 509.897,Z 452.972,A -85,B 0,C 180,E1 -5595.242,E2 -5595.242} C_VEL
LIN {X 0,Y 509.892,Z 452.97,A -85,B 0,C 180,E1 -5598.001,E2 -5598.001} C_VEL
LIN {X 0,Y 509.854,Z 452.975,A -85,B 0,C 180,E1 -5601.002,E2 -5601.002} C_VEL
LIN {X 0,Y 509.868,Z 452.975,A -85,B 0,C 180,E1 -5604.426,E2 -5604.426} C_VEL
LIN {X 0,Y 509.889,Z 452.97,A -85,B 0,C 180,E1 -5607.056,E2 -5607.056} C_VEL
LIN {X 0,Y 509.86,Z 452.976,A -85,B 0,C 180,E1 -5609.751,E2 -5609.751} C_VEL
LIN {X 0,Y 509.878,Z 452.973,A -85,B 0,C 180,E1 -5612.775,E2 -5612.775} C_VEL
LIN {X 0,Y 509.844,Z 452.978,A -85,B 0,C 180,E1 -5615.581,E2 -5615.581} C_VEL
LIN {X 0,Y 509.853,Z 452.976,A -85,B 0,C 180,E1 -5618.338,E2 -5618.338} C_VEL
LIN {X 0,Y 509.861,Z 452.974,A -85,B 0,C 180,E1 -5621.425,E2 -5621.425} C_VEL
LIN {X 0,Y 509.86,Z 452.976,A -85,B 0,C 180,E1 -5624.668,E2 -5624.668} C_VEL
LIN {X 0,Y 509.859,Z 452.978,A -85,B 0,C 180,E1 -5628.104,E2 -5628.104} C_VEL
LIN {X 0,Y 509.85,Z 452.976,A -85,B 0,C 180,E1 -5630.648,E2 -5630.648} C_VEL
LIN {X 0,Y 509.833,Z 452.977,A -85,B 0,C 180,E1 -5633.736,E2 -5633.736} C_VEL
LIN {X 0,Y 509.167,Z 453.064,A -85,B 0,C 180,E1 -5634.396,E2 -5634.396} C_VEL
LIN {X 0,Y 506.352,Z 453.412,A -85,B 0,C 180,E1 -5635.468,E2 -5635.468} C_VEL
LIN {X 0,Y 503.96,Z 453.71,A -85,B 0,C 180,E1 -5636.331,E2 -5636.331} C_VEL
LIN {X 0,Y 502.91,Z 453.84,A -85,B 0,C 180,E1 -5636.998,E2 -5636.998} C_VEL
LIN {X 0,Y 502.812,Z 453.851,A -85,B 0,C 180,E1 -5637.223,E2 -5637.223} C_VEL
LIN {X 0,Y 502.819,Z 453.852,A -85,B 0,C 180,E1 -5640.065,E2 -5640.065} C_VEL
LIN {X 0,Y 502.835,Z 453.85,A -85,B 0,C 180,E1 -5642.533,E2 -5642.533} C_VEL
LIN {X 0,Y 502.831,Z 453.852,A -85,B 0,C 180,E1 -5645.299,E2 -5645.299} C_VEL
LIN {X 0,Y 502.785,Z 453.855,A -85,B 0,C 180,E1 -5647.827,E2 -5647.827} C_VEL
LIN {X 0,Y 502.829,Z 453.85,A -85,B 0,C 180,E1 -5650.4,E2 -5650.4} C_VEL
LIN {X 0,Y 502.825,Z 453.853,A -85,B 0,C 180,E1 -5652.931,E2 -5652.931} C_VEL
LIN {X 0,Y 502.85,Z 453.847,A -85,B 0,C 180,E1 -5655.429,E2 -5655.429} C_VEL
LIN {X 0,Y 502.883,Z 453.843,A -85,B 0,C 180,E1 -5658.717,E2 -5658.717} C_VEL
LIN {X 0,Y 502.906,Z 453.841,A -85,B 0,C 180,E1 -5661.967,E2 -5661.967} C_VEL
LIN {X 0,Y 502.931,Z 453.838,A -85,B 0,C 180,E1 -5664.387,E2 -5664.387} C_VEL
LIN {X 0,Y 503.03,Z 453.826,A -85,B 0,C 180,E1 -5667.598,E2 -5667.598} C_VEL
LIN {X 0,Y 503.033,Z 453.827,A -85,B 0,C 180,E1 -5670,E2 -5670} C_VEL
LIN {X 0,Y 503.03,Z 453.825,A -85,B 0,C 180,E1 -5672.402,E2 -5672.402} C_VEL
LIN {X 0,Y 502.934,Z 453.84,A -85,B 0,C 180,E1 -5676.419,E2 -5676.419} C_VEL
LIN {X 0,Y 502.843,Z 453.852,A -85,B 0,C 180,E1 -5679.655,E2 -5679.655} C_VEL
LIN {X 0,Y 502.852,Z 453.848,A -85,B 0,C 180,E1 -5682.102,E2 -5682.102} C_VEL
LIN {X 0,Y 502.854,Z 453.846,A -85,B 0,C 180,E1 -5685.4,E2 -5685.4} C_VEL
LIN {X 0,Y 502.846,Z 453.848,A -85,B 0,C 180,E1 -5688.12,E2 -5688.12} C_VEL
LIN {X 0,Y 502.834,Z 453.852,A -85,B 0,C 180,E1 -5690.536,E2 -5690.536} C_VEL
LIN {X 0,Y 502.797,Z 453.852,A -85,B 0,C 180,E1 -5693.041,E2 -5693.041} C_VEL
LIN {X 0,Y 502.845,Z 453.849,A -85,B 0,C 180,E1 -5695.675,E2 -5695.675} C_VEL
LIN {X 0,Y 502.845,Z 453.85,A -85,B 0,C 180,E1 -5698.373,E2 -5698.373} C_VEL
LIN {X 0,Y 502.798,Z 453.858,A -85,B 0,C 180,E1 -5701.499,E2 -5701.499} C_VEL
LIN {X 0,Y 502.809,Z 453.853,A -85,B 0,C 180,E1 -5703.994,E2 -5703.994} C_VEL
LIN {X 0,Y 502.782,Z 453.855,A -85,B 0,C 180,E1 -5707.178,E2 -5707.178} C_VEL
LIN {X 0,Y 502.793,Z 453.855,A -85,B 0,C 180,E1 -5710.015,E2 -5710.015} C_VEL
LIN {X 0,Y 502.807,Z 453.856,A -85,B 0,C 180,E1 -5712.199,E2 -5712.199} C_VEL
LIN {X 0,Y 502.79,Z 453.858,A -85,B 0,C 180,E1 -5715.47,E2 -5715.47} C_VEL
LIN {X 0,Y 502.825,Z 453.852,A -85,B 0,C 180,E1 -5718.934,E2 -5718.934} C_VEL
LIN {X 0,Y 502.794,Z 453.855,A -85,B 0,C 180,E1 -5722.046,E2 -5722.046} C_VEL
LIN {X 0,Y 502.686,Z 453.871,A -85,B 0,C 180,E1 -5725.025,E2 -5725.025} C_VEL
LIN {X 0,Y 502.396,Z 453.908,A -85,B 0,C 180,E1 -5727.887,E2 -5727.887} C_VEL
LIN {X 0,Y 502.351,Z 454.46,A -85,B 0,C 180,E1 -5728.826,E2 -5728.826} C_VEL
LIN {X 0,Y 502.306,Z 457.658,A -85,B 0,C 180,E1 -5731.82,E2 -5731.82} C_VEL
LIN {X 0,Y 502.281,Z 460.355,A -85,B 0,C 180,E1 -5734.293,E2 -5734.293} C_VEL
LIN {X 0,Y 502.201,Z 463.803,A -85,B 0,C 180,E1 -5737.463,E2 -5737.463} C_VEL
LIN {X 0,Y 502.194,Z 467.043,A -85,B 0,C 180,E1 -5740.374,E2 -5740.374} C_VEL
LIN {X 0,Y 502.144,Z 469.878,A -85,B 0,C 180,E1 -5742.907,E2 -5742.907} C_VEL
LIN {X 0,Y 502.178,Z 473.388,A -85,B 0,C 180,E1 -5745.836,E2 -5745.836} C_VEL
LIN {X 0,Y 504.597,Z 485.663,A -85,B 0,C 180,E1 -5746.252,E2 -5746.252} C_VEL
LIN {X 0,Y 504.362,Z 498.18,A -85,B 0,C 180,E1 -5746.759,E2 -5746.759} C_VEL
LIN {X 0,Y 504.018,Z 510.047,A -85,B 0,C 180,E1 -5747.403,E2 -5747.403} C_VEL
LIN {X 0,Y 503.662,Z 521.709,A -85,B 0,C 180,E1 -5748.224,E2 -5748.224} C_VEL
LIN {X 0,Y 503.348,Z 532.05,A -85,B 0,C 180,E1 -5749.135,E2 -5749.135} C_VEL
LIN {X 0,Y 503.014,Z 541.36,A -85,B 0,C 180,E1 -5750.145,E2 -5750.145} C_VEL
LIN {X 0,Y 502.715,Z 550.346,A -85,B 0,C 180,E1 -5751.356,E2 -5751.356} C_VEL
LIN {X 0,Y 502.475,Z 557.594,A -85,B 0,C 180,E1 -5752.566,E2 -5752.566} C_VEL
LIN {X 0,Y 502.349,Z 564.197,A -85,B 0,C 180,E1 -5753.977,E2 -5753.977} C_VEL
LIN {X 0,Y 502.13,Z 568.565,A -85,B 0,C 180,E1 -5755.183,E2 -5755.183} C_VEL
LIN {X 0,Y 502.236,Z 570.861,A -85,B 0,C 180,E1 -5755.988,E2 -5755.988} C_VEL
LIN {X 0,Y 502.125,Z 572.753,A -85,B 0,C 180,E1 -5756.79,E2 -5756.79} C_VEL
LIN {X 0,Y 502.121,Z 574.174,A -85,B 0,C 180,E1 -5757.593,E2 -5757.593} C_VEL
LIN {X 0,Y 501.991,Z 575.818,A -85,B 0,C 180,E1 -5759.198,E2 -5759.198} C_VEL
LIN {X 0,Y 501.982,Z 576.07,A -85,B 0,C 180,E1 -5760,E2 -5760} C_VEL
LIN {X 0,Y 501.991,Z 575.893,A -85,B 0,C 180,E1 -5760.802,E2 -5760.802} C_VEL
LIN {X 0,Y 502.121,Z 574.355,A -85,B 0,C 180,E1 -5762.406,E2 -5762.406} C_VEL
LIN {X 0,Y 502.137,Z 573.009,A -85,B 0,C 180,E1 -5763.209,E2 -5763.209} C_VEL
LIN {X 0,Y 502.21,Z 570.152,A -85,B 0,C 180,E1 -5764.414,E2 -5764.414} C_VEL
LIN {X 0,Y 502.285,Z 566.27,A -85,B 0,C 180,E1 -5765.621,E2 -5765.621} C_VEL
LIN {X 0,Y 502.409,Z 560.371,A -85,B 0,C 180,E1 -5767.01,E2 -5767.01} C_VEL
LIN {X 0,Y 502.609,Z 553.69,A -85,B 0,C 180,E1 -5768.24,E2 -5768.24} C_VEL
LIN {X 0,Y 502.841,Z 545.506,A -85,B 0,C 180,E1 -5769.452,E2 -5769.452} C_VEL
LIN {X 0,Y 503.134,Z 537.092,A -85,B 0,C 180,E1 -5770.462,E2 -5770.462} C_VEL
LIN {X 0,Y 503.579,Z 526.677,A -85,B 0,C 180,E1 -5771.471,E2 -5771.471} C_VEL
LIN {X 0,Y 503.897,Z 515.085,A -85,B 0,C 180,E1 -5772.374,E2 -5772.374} C_VEL
LIN {X 0,Y 504.235,Z 503.178,A -85,B 0,C 180,E1 -5773.091,E2 -5773.091} C_VEL
LIN {X 0,Y 504.535,Z 491.039,A -85,B 0,C 180,E1 -5773.647,E2 -5773.647} C_VEL
LIN {X 0,Y 504.386,Z 484.729,A -85,B 0,C 180,E1 -5773.882,E2 -5773.882} C_VEL
LIN {X 0,Y 502.555,Z 475.641,A -85,B 0,C 180,E1 -5774.192,E2 -5774.192} C_VEL
LIN {X 0,Y 502.227,Z 474.068,A -85,B 0,C 180,E1 -5774.253,E2 -5774.253} C_VEL
LIN {X 0,Y 502.235,Z 471.143,A -85,B 0,C 180,E1 -5777.089,E2 -5777.089} C_VEL
LIN {X 0,Y 502.353,Z 467.772,A -85,B 0,C 180,E1 -5780.472,E2 -5780.472} C_VEL
LIN {X 0,Y 502.388,Z 465.291,A -85,B 0,C 180,E1 -5783.06,E2 -5783.06} C_VEL
LIN {X 0,Y 502.485,Z 462.835,A -85,B 0,C 180,E1 -5785.695,E2 -5785.695} C_VEL
LIN {X 0,Y 502.592,Z 460.437,A -85,B 0,C 180,E1 -5788.388,E2 -5788.388} C_VEL
LIN {X 0,Y 502.722,Z 457.863,A -85,B 0,C 180,E1 -5791.485,E2 -5791.485} C_VEL
LIN {X 0,Y 502.847,Z 455.546,A -85,B 0,C 180,E1 -5794.451,E2 -5794.451} C_VEL
LIN {X 0,Y 502.766,Z 453.862,A -85,B 0,C 180,E1 -5797.175,E2 -5797.175} C_VEL
LIN {X 0,Y 502.791,Z 453.859,A -85,B 0,C 180,E1 -5800.015,E2 -5800.015} C_VEL
LIN {X 0,Y 502.806,Z 453.856,A -85,B 0,C 180,E1 -5802.199,E2 -5802.199} C_VEL
LIN {X 0,Y 502.804,Z 453.857,A -85,B 0,C 180,E1 -5805.468,E2 -5805.468} C_VEL
LIN {X 0,Y 502.833,Z 454.041,A -85,B 0,C 180,E1 -5807.864,E2 -5807.864} C_VEL
LIN {X 0,Y 503.317,Z 456.509,A -85,B 0,C 180,E1 -5810.173,E2 -5810.173} C_VEL
LIN {X 0,Y 503.925,Z 460.226,A -85,B 0,C 180,E1 -5812.651,E2 -5812.651} C_VEL
LIN {X 0,Y 504.246,Z 464.039,A -85,B 0,C 180,E1 -5814.661,E2 -5814.661} C_VEL
LIN {X 0,Y 503.822,Z 469.458,A -85,B 0,C 180,E1 -5817.042,E2 -5817.042} C_VEL
LIN {X 0,Y 503.441,Z 476.836,A -85,B 0,C 180,E1 -5819.942,E2 -5819.942} C_VEL
LIN {X 0,Y 503.111,Z 485.386,A -85,B 0,C 180,E1 -5823,E2 -5823} C_VEL
LIN {X 0,Y 502.888,Z 493.376,A -85,B 0,C 180,E1 -5825.68,E2 -5825.68} C_VEL
LIN {X 0,Y 502.697,Z 502.752,A -85,B 0,C 180,E1 -5828.685,E2 -5828.685} C_VEL
LIN {X 0,Y 502.537,Z 512.488,A -85,B 0,C 180,E1 -5831.702,E2 -5831.702} C_VEL
LIN {X 0,Y 502.451,Z 522.799,A -85,B 0,C 180,E1 -5834.826,E2 -5834.826} C_VEL
LIN {X 0,Y 502.388,Z 525.696,A -85,B 0,C 180,E1 -5835.7,E2 -5835.7} C_VEL
LIN {X 0,Y 504.536,Z 541.448,A -85,B 0,C 180,E1 -5836.173,E2 -5836.173} C_VEL
LIN {X 0,Y 504.197,Z 554.888,A -85,B 0,C 180,E1 -5836.703,E2 -5836.703} C_VEL
LIN {X 0,Y 503.858,Z 566.946,A -85,B 0,C 180,E1 -5837.349,E2 -5837.349} C_VEL
LIN {X 0,Y 503.522,Z 578.13,A -85,B 0,C 180,E1 -5838.119,E2 -5838.119} C_VEL
LIN {X 0,Y 503.181,Z 588.77,A -85,B 0,C 180,E1 -5839.029,E2 -5839.029} C_VEL
LIN {X 0,Y 502.888,Z 597.483,A -85,B 0,C 180,E1 -5839.939,E2 -5839.939} C_VEL
LIN {X 0,Y 502.661,Z 605.526,A -85,B 0,C 180,E1 -5840.95,E2 -5840.95} C_VEL
LIN {X 0,Y 502.417,Z 613.382,A -85,B 0,C 180,E1 -5842.161,E2 -5842.161} C_VEL
LIN {X 0,Y 502.263,Z 620.061,A -85,B 0,C 180,E1 -5843.455,E2 -5843.455} C_VEL
LIN {X 0,Y 502.183,Z 625.414,A -85,B 0,C 180,E1 -5844.781,E2 -5844.781} C_VEL
LIN {X 0,Y 502.166,Z 629.09,A -85,B 0,C 180,E1 -5845.987,E2 -5845.987} C_VEL
LIN {X 0,Y 502.121,Z 630.99,A -85,B 0,C 180,E1 -5846.79,E2 -5846.79} C_VEL
LIN {X 0,Y 502.12,Z 632.412,A -85,B 0,C 180,E1 -5847.593,E2 -5847.593} C_VEL
LIN {X 0,Y 501.99,Z 634.043,A -85,B 0,C 180,E1 -5849.198,E2 -5849.198} C_VEL
LIN {X 0,Y 501.98,Z 634.27,A -85,B 0,C 180,E1 -5850,E2 -5850} C_VEL
LIN {X 0,Y 502.036,Z 633.45,A -85,B 0,C 180,E1 -5851.604,E2 -5851.604} C_VEL
LIN {X 0,Y 502.12,Z 632.454,A -85,B 0,C 180,E1 -5852.406,E2 -5852.406} C_VEL
LIN {X 0,Y 502.121,Z 631.046,A -85,B 0,C 180,E1 -5853.209,E2 -5853.209} C_VEL
LIN {X 0,Y 502.125,Z 628.084,A -85,B 0,C 180,E1 -5854.415,E2 -5854.415} C_VEL
LIN {X 0,Y 502.238,Z 624.075,A -85,B 0,C 180,E1 -5855.621,E2 -5855.621} C_VEL
LIN {X 0,Y 502.332,Z 617.996,A -85,B 0,C 180,E1 -5857.011,E2 -5857.011} C_VEL
LIN {X 0,Y 502.499,Z 611.147,A -85,B 0,C 180,E1 -5858.242,E2 -5858.242} C_VEL
LIN {X 0,Y 502.73,Z 602.779,A -85,B 0,C 180,E1 -5859.454,E2 -5859.454} C_VEL
LIN {X 0,Y 503.013,Z 594.183,A -85,B 0,C 180,E1 -5860.465,E2 -5860.465} C_VEL
LIN {X 0,Y 503.38,Z 583.581,A -85,B 0,C 180,E1 -5861.476,E2 -5861.476} C_VEL
LIN {X 0,Y 503.703,Z 573.697,A -85,B 0,C 180,E1 -5862.243,E2 -5862.243} C_VEL
LIN {X 0,Y 504.07,Z 561.632,A -85,B 0,C 180,E1 -5862.992,E2 -5862.992} C_VEL
LIN {X 0,Y 504.418,Z 549.799,A -85,B 0,C 180,E1 -5863.547,E2 -5863.547} C_VEL
LIN {X 0,Y 504.43,Z 539.889,A -85,B 0,C 180,E1 -5863.906,E2 -5863.906} C_VEL
LIN {X 0,Y 502.484,Z 527.152,A -85,B 0,C 180,E1 -5864.271,E2 -5864.271} C_VEL
LIN {X 0,Y 502.414,Z 526.388,A -85,B 0,C 180,E1 -5864.299,E2 -5864.299} C_VEL
LIN {X 0,Y 502.547,Z 517.456,A -85,B 0,C 180,E1 -5867.078,E2 -5867.078} C_VEL
LIN {X 0,Y 502.715,Z 508.145,A -85,B 0,C 180,E1 -5870.03,E2 -5870.03} C_VEL
LIN {X 0,Y 502.915,Z 498.855,A -85,B 0,C 180,E1 -5873.035,E2 -5873.035} C_VEL
LIN {X 0,Y 503.221,Z 489.653,A -85,B 0,C 180,E1 -5876.099,E2 -5876.099} C_VEL
LIN {X 0,Y 503.447,Z 481.796,A -85,B 0,C 180,E1 -5878.79,E2 -5878.79} C_VEL
LIN {X 0,Y 503.838,Z 473.57,A -85,B 0,C 180,E1 -5881.692,E2 -5881.692} C_VEL
LIN {X 0,Y 504.167,Z 464.936,A -85,B 0,C 180,E1 -5884.857,E2 -5884.857} C_VEL
LIN {X 0,Y 504.025,Z 460.898,A -85,B 0,C 180,E1 -5886.403,E2 -5886.403} C_VEL
LIN {X 0,Y 502.827,Z 453.854,A -85,B 0,C 180,E1 -5889.361,E2 -5889.361} C_VEL
LIN {X 0,Y 502.804,Z 453.854,A -85,B 0,C 180,E1 -5892.199,E2 -5892.199} C_VEL
LIN {X 0,Y 502.803,Z 453.853,A -85,B 0,C 180,E1 -5895.468,E2 -5895.468} C_VEL
LIN {X 0,Y 502.832,Z 453.852,A -85,B 0,C 180,E1 -5897.864,E2 -5897.864} C_VEL
LIN {X 0,Y 502.802,Z 453.855,A -85,B 0,C 180,E1 -5901.024,E2 -5901.024} C_VEL
LIN {X 0,Y 502.777,Z 453.859,A -85,B 0,C 180,E1 -5904.169,E2 -5904.169} C_VEL
LIN {X 0,Y 502.834,Z 453.853,A -85,B 0,C 180,E1 -5906.993,E2 -5906.993} C_VEL
LIN {X 0,Y 502.816,Z 453.854,A -85,B 0,C 180,E1 -5910.065,E2 -5910.065} C_VEL
LIN {X 0,Y 502.836,Z 453.849,A -85,B 0,C 180,E1 -5912.533,E2 -5912.533} C_VEL
LIN {X 0,Y 502.825,Z 453.849,A -85,B 0,C 180,E1 -5915.3,E2 -5915.3} C_VEL
LIN {X 0,Y 502.782,Z 453.858,A -85,B 0,C 180,E1 -5917.827,E2 -5917.827} C_VEL
LIN {X 0,Y 502.828,Z 453.85,A -85,B 0,C 180,E1 -5920.4,E2 -5920.4} C_VEL
LIN {X 0,Y 502.837,Z 453.85,A -85,B 0,C 180,E1 -5922.932,E2 -5922.932} C_VEL
LIN {X 0,Y 502.848,Z 453.85,A -85,B 0,C 180,E1 -5925.429,E2 -5925.429} C_VEL
LIN {X 0,Y 502.879,Z 453.847,A -85,B 0,C 180,E1 -5928.717,E2 -5928.717} C_VEL
LIN {X 0,Y 502.904,Z 453.843,A -85,B 0,C 180,E1 -5931.967,E2 -5931.967} C_VEL
LIN {X 0,Y 502.94,Z 453.836,A -85,B 0,C 180,E1 -5934.387,E2 -5934.387} C_VEL
LIN {X 0,Y 503.026,Z 453.824,A -85,B 0,C 180,E1 -5937.598,E2 -5937.598} C_VEL
LIN {X 0,Y 503.03,Z 453.828,A -85,B 0,C 180,E1 -5940,E2 -5940} C_VEL
LIN {X 0,Y 503.026,Z 453.826,A -85,B 0,C 180,E1 -5942.402,E2 -5942.402} C_VEL
LIN {X 0,Y 502.94,Z 453.836,A -85,B 0,C 180,E1 -5945.614,E2 -5945.614} C_VEL
LIN {X 0,Y 502.905,Z 453.842,A -85,B 0,C 180,E1 -5948.033,E2 -5948.033} C_VEL
LIN {X 0,Y 502.88,Z 453.842,A -85,B 0,C 180,E1 -5951.283,E2 -5951.283} C_VEL
LIN {X 0,Y 502.848,Z 453.848,A -85,B 0,C 180,E1 -5954.571,E2 -5954.571} C_VEL
LIN {X 0,Y 502.865,Z 453.845,A -85,B 0,C 180,E1 -5957.907,E2 -5957.907} C_VEL
LIN {X 0,Y 502.832,Z 453.85,A -85,B 0,C 180,E1 -5960.536,E2 -5960.536} C_VEL
LIN {X 0,Y 502.794,Z 453.857,A -85,B 0,C 180,E1 -5963.041,E2 -5963.041} C_VEL
LIN {X 0,Y 502.843,Z 453.847,A -85,B 0,C 180,E1 -5965.676,E2 -5965.676} C_VEL
LIN {X 0,Y 502.844,Z 453.849,A -85,B 0,C 180,E1 -5968.373,E2 -5968.373} C_VEL
LIN {X 0,Y 502.797,Z 453.854,A -85,B 0,C 180,E1 -5971.499,E2 -5971.499} C_VEL
LIN {X 0,Y 502.808,Z 453.854,A -85,B 0,C 180,E1 -5974.445,E2 -5974.445} C_VEL
LIN {X 0,Y 502.784,Z 453.858,A -85,B 0,C 180,E1 -5977.179,E2 -5977.179} C_VEL
LIN {X 0,Y 502.791,Z 453.856,A -85,B 0,C 180,E1 -5980.015,E2 -5980.015} C_VEL
LIN {X 0,Y 502.806,Z 453.855,A -85,B 0,C 180,E1 -5982.199,E2 -5982.199} C_VEL
LIN {X 0,Y 502.804,Z 453.854,A -85,B 0,C 180,E1 -5985.468,E2 -5985.468} C_VEL
LIN {X 0,Y 502.823,Z 453.85,A -85,B 0,C 180,E1 -5988.934,E2 -5988.934} C_VEL
LIN {X 0,Y 502.797,Z 453.854,A -85,B 0,C 180,E1 -5992.046,E2 -5992.046} C_VEL
LIN {X 0,Y 502.812,Z 453.85,A -85,B 0,C 180,E1 -5995.035,E2 -5995.035} C_VEL
LIN {X 0,Y 502.812,Z 453.851,A -85,B 0,C 180,E1 -5997.223,E2 -5997.223} C_VEL
LIN {X 0,Y 502.11,Z 453.941,A -85,B 0,C 180,E1 -5997.892,E2 -5997.892} C_VEL
LIN {X 0,Y 499.246,Z 454.299,A -85,B 0,C 180,E1 -5998.978,E2 -5998.978} C_VEL
LIN {X 0,Y 496.852,Z 454.596,A -85,B 0,C 180,E1 -5999.853,E2 -5999.853} C_VEL
LIN {X 0,Y 495.835,Z 454.725,A -85,B 0,C 180,E1 -6000.528,E2 -6000.528} C_VEL
LIN {X 0,Y 495.757,Z 454.729,A -85,B 0,C 180,E1 -6000.757,E2 -6000.757} C_VEL
LIN {X 0,Y 495.795,Z 454.729,A -85,B 0,C 180,E1 -6003.932,E2 -6003.932} C_VEL
LIN {X 0,Y 495.765,Z 454.731,A -85,B 0,C 180,E1 -6007.139,E2 -6007.139} C_VEL
LIN {X 0,Y 495.776,Z 454.732,A -85,B 0,C 180,E1 -6010.11,E2 -6010.11} C_VEL
LIN {X 0,Y 495.77,Z 454.731,A -85,B 0,C 180,E1 -6012.681,E2 -6012.681} C_VEL
LIN {X 0,Y 495.795,Z 454.726,A -85,B 0,C 180,E1 -6015.217,E2 -6015.217} C_VEL
LIN {X 0,Y 495.857,Z 454.718,A -85,B 0,C 180,E1 -6018.555,E2 -6018.555} C_VEL
LIN {X 0,Y 495.878,Z 454.716,A -85,B 0,C 180,E1 -6021.852,E2 -6021.852} C_VEL
LIN {X 0,Y 495.842,Z 454.72,A -85,B 0,C 180,E1 -6025.122,E2 -6025.122} C_VEL
LIN {X 0,Y 495.998,Z 454.702,A -85,B 0,C 180,E1 -6027.564,E2 -6027.564} C_VEL
LIN {X 0,Y 496.004,Z 454.702,A -85,B 0,C 180,E1 -6030,E2 -6030} C_VEL
LIN {X 0,Y 495.998,Z 454.701,A -85,B 0,C 180,E1 -6032.436,E2 -6032.436} C_VEL
LIN {X 0,Y 495.9,Z 454.713,A -85,B 0,C 180,E1 -6035.694,E2 -6035.694} C_VEL
LIN {X 0,Y 495.842,Z 454.723,A -85,B 0,C 180,E1 -6038.149,E2 -6038.149} C_VEL
LIN {X 0,Y 495.857,Z 454.721,A -85,B 0,C 180,E1 -6041.445,E2 -6041.445} C_VEL
LIN {X 0,Y 495.796,Z 454.725,A -85,B 0,C 180,E1 -6044.783,E2 -6044.783} C_VEL
LIN {X 0,Y 495.786,Z 454.729,A -85,B 0,C 180,E1 -6047.319,E2 -6047.319} C_VEL
LIN {X 0,Y 495.776,Z 454.729,A -85,B 0,C 180,E1 -6049.89,E2 -6049.89} C_VEL
LIN {X 0,Y 495.765,Z 454.728,A -85,B 0,C 180,E1 -6052.861,E2 -6052.861} C_VEL
LIN {X 0,Y 495.796,Z 454.726,A -85,B 0,C 180,E1 -6056.068,E2 -6056.068} C_VEL
LIN {X 0,Y 495.777,Z 454.728,A -85,B 0,C 180,E1 -6058.815,E2 -6058.815} C_VEL
LIN {X 0,Y 495.76,Z 454.733,A -85,B 0,C 180,E1 -6061.725,E2 -6061.725} C_VEL
LIN {X 0,Y 495.774,Z 454.731,A -85,B 0,C 180,E1 -6064.694,E2 -6064.694} C_VEL
LIN {X 0,Y 495.734,Z 454.736,A -85,B 0,C 180,E1 -6067.561,E2 -6067.561} C_VEL
LIN {X 0,Y 495.771,Z 454.731,A -85,B 0,C 180,E1 -6070.7,E2 -6070.7} C_VEL
LIN {X 0,Y 495.732,Z 454.737,A -85,B 0,C 180,E1 -6074.002,E2 -6074.002} C_VEL
LIN {X 0,Y 495.73,Z 454.737,A -85,B 0,C 180,E1 -6077.117,E2 -6077.117} C_VEL
LIN {X 0,Y 495.763,Z 454.733,A -85,B 0,C 180,E1 -6079.953,E2 -6079.953} C_VEL
LIN {X 0,Y 495.721,Z 454.734,A -85,B 0,C 180,E1 -6082.555,E2 -6082.555} C_VEL
LIN {X 0,Y 495.639,Z 454.749,A -85,B 0,C 180,E1 -6085.445,E2 -6085.445} C_VEL
LIN {X 0,Y 495.293,Z 454.793,A -85,B 0,C 180,E1 -6088.362,E2 -6088.362} C_VEL
LIN {X 0,Y 495.229,Z 457.584,A -85,B 0,C 180,E1 -6091.15,E2 -6091.15} C_VEL
LIN {X 0,Y 495.235,Z 460.54,A -85,B 0,C 180,E1 -6093.9,E2 -6093.9} C_VEL
LIN {X 0,Y 495.143,Z 463.452,A -85,B 0,C 180,E1 -6096.582,E2 -6096.582} C_VEL
LIN {X 0,Y 495.123,Z 467.291,A -85,B 0,C 180,E1 -6100.082,E2 -6100.082} C_VEL
LIN {X 0,Y 495.085,Z 470.167,A -85,B 0,C 180,E1 -6102.656,E2 -6102.656} C_VEL
LIN {X 0,Y 495.066,Z 473.503,A -85,B 0,C 180,E1 -6105.615,E2 -6105.615} C_VEL
LIN {X 0,Y 497.653,Z 486.526,A -85,B 0,C 180,E1 -6106.083,E2 -6106.083} C_VEL
LIN {X 0,Y 497.414,Z 499.426,A -85,B 0,C 180,E1 -6106.622,E2 -6106.622} C_VEL
LIN {X 0,Y 497.014,Z 512.051,A -85,B 0,C 180,E1 -6107.342,E2 -6107.342} C_VEL
LIN {X 0,Y 496.692,Z 523.207,A -85,B 0,C 180,E1 -6108.16,E2 -6108.16} C_VEL
LIN {X 0,Y 496.358,Z 533.33,A -85,B 0,C 180,E1 -6109.083,E2 -6109.083} C_VEL
LIN {X 0,Y 495.946,Z 543.256,A -85,B 0,C 180,E1 -6110.209,E2 -6110.209} C_VEL
LIN {X 0,Y 495.661,Z 552.004,A -85,B 0,C 180,E1 -6111.438,E2 -6111.438} C_VEL
LIN {X 0,Y 495.405,Z 558.977,A -85,B 0,C 180,E1 -6112.664,E2 -6112.664} C_VEL
LIN {X 0,Y 495.29,Z 564.546,A -85,B 0,C 180,E1 -6113.891,E2 -6113.891} C_VEL
LIN {X 0,Y 495.058,Z 568.933,A -85,B 0,C 180,E1 -6115.114,E2 -6115.114} C_VEL
LIN {X 0,Y 495.17,Z 571.24,A -85,B 0,C 180,E1 -6115.93,E2 -6115.93} C_VEL
LIN {X 0,Y 495.051,Z 573.141,A -85,B 0,C 180,E1 -6116.744,E2 -6116.744} C_VEL
LIN {X 0,Y 495.054,Z 574.569,A -85,B 0,C 180,E1 -6117.559,E2 -6117.559} C_VEL
LIN {X 0,Y 494.911,Z 576.227,A -85,B 0,C 180,E1 -6119.186,E2 -6119.186} C_VEL
LIN {X 0,Y 494.899,Z 576.482,A -85,B 0,C 180,E1 -6120,E2 -6120} C_VEL
LIN {X 0,Y 494.911,Z 576.307,A -85,B 0,C 180,E1 -6120.814,E2 -6120.814} C_VEL
LIN {X 0,Y 495.055,Z 574.77,A -85,B 0,C 180,E1 -6122.441,E2 -6122.441} C_VEL
LIN {X 0,Y 495.062,Z 573.423,A -85,B 0,C 180,E1 -6123.255,E2 -6123.255} C_VEL
LIN {X 0,Y 495.14,Z 570.561,A -85,B 0,C 180,E1 -6124.477,E2 -6124.477} C_VEL
LIN {X 0,Y 495.231,Z 566.67,A -85,B 0,C 180,E1 -6125.701,E2 -6125.701} C_VEL
LIN {X 0,Y 495.37,Z 560.753,A -85,B 0,C 180,E1 -6127.11,E2 -6127.11} C_VEL
LIN {X 0,Y 495.604,Z 554.053,A -85,B 0,C 180,E1 -6128.358,E2 -6128.358} C_VEL
LIN {X 0,Y 495.85,Z 545.85,A -85,B 0,C 180,E1 -6129.587,E2 -6129.587} C_VEL
LIN {X 0,Y 496.154,Z 537.403,A -85,B 0,C 180,E1 -6130.611,E2 -6130.611} C_VEL
LIN {X 0,Y 496.637,Z 526.961,A -85,B 0,C 180,E1 -6131.634,E2 -6131.634} C_VEL
LIN {X 0,Y 496.957,Z 515.332,A -85,B 0,C 180,E1 -6132.55,E2 -6132.55} C_VEL
LIN {X 0,Y 497.325,Z 503.389,A -85,B 0,C 180,E1 -6133.276,E2 -6133.276} C_VEL
LIN {X 0,Y 497.639,Z 491.221,A -85,B 0,C 180,E1 -6133.839,E2 -6133.839} C_VEL
LIN {X 0,Y 497.429,Z 485.26,A -85,B 0,C 180,E1 -6134.067,E2 -6134.067} C_VEL
LIN {X 0,Y 495.502,Z 476.174,A -85,B 0,C 180,E1 -6134.388,E2 -6134.388} C_VEL
LIN {X 0,Y 495.181,Z 474.595,A -85,B 0,C 180,E1 -6134.46,E2 -6134.46} C_VEL
LIN {X 0,Y 495.194,Z 471.655,A -85,B 0,C 180,E1 -6137.34,E2 -6137.34} C_VEL
LIN {X 0,Y 495.289,Z 468.29,A -85,B 0,C 180,E1 -6140.778,E2 -6140.778} C_VEL
LIN {X 0,Y 495.354,Z 465.817,A -85,B 0,C 180,E1 -6143.407,E2 -6143.407} C_VEL
LIN {X 0,Y 495.448,Z 463.381,A -85,B 0,C 180,E1 -6146.087,E2 -6146.087} C_VEL
LIN {X 0,Y 495.574,Z 461.028,A -85,B 0,C 180,E1 -6148.827,E2 -6148.827} C_VEL
LIN {X 0,Y 495.714,Z 458.714,A -85,B 0,C 180,E1 -6151.717,E2 -6151.717} C_VEL
LIN {X 0,Y 495.846,Z 456.512,A -85,B 0,C 180,E1 -6154.706,E2 -6154.706} C_VEL
LIN {X 0,Y 495.74,Z 454.862,A -85,B 0,C 180,E1 -6157.561,E2 -6157.561} C_VEL
LIN {X 0,Y 495.762,Z 454.734,A -85,B 0,C 180,E1 -6160.047,E2 -6160.047} C_VEL
LIN {X 0,Y 495.736,Z 454.737,A -85,B 0,C 180,E1 -6162.882,E2 -6162.882} C_VEL
LIN {X 0,Y 495.737,Z 454.738,A -85,B 0,C 180,E1 -6165.999,E2 -6165.999} C_VEL
LIN {X 0,Y 495.839,Z 455.333,A -85,B 0,C 180,E1 -6167.481,E2 -6167.481} C_VEL
LIN {X 0,Y 496.308,Z 457.731,A -85,B 0,C 180,E1 -6169.878,E2 -6169.878} C_VEL
LIN {X 0,Y 496.914,Z 461.276,A -85,B 0,C 180,E1 -6172.375,E2 -6172.375} C_VEL
LIN {X 0,Y 497.29,Z 465.332,A -85,B 0,C 180,E1 -6174.589,E2 -6174.589} C_VEL
LIN {X 0,Y 496.846,Z 470.664,A -85,B 0,C 180,E1 -6177.018,E2 -6177.018} C_VEL
LIN {X 0,Y 496.458,Z 477.348,A -85,B 0,C 180,E1 -6179.716,E2 -6179.716} C_VEL
LIN {X 0,Y 496.08,Z 486.433,A -85,B 0,C 180,E1 -6183.041,E2 -6183.041} C_VEL
LIN {X 0,Y 495.82,Z 494.299,A -85,B 0,C 180,E1 -6185.728,E2 -6185.728} C_VEL
LIN {X 0,Y 495.633,Z 503.702,A -85,B 0,C 180,E1 -6188.802,E2 -6188.802} C_VEL
LIN {X 0,Y 495.444,Z 513.454,A -85,B 0,C 180,E1 -6191.882,E2 -6191.882} C_VEL
LIN {X 0,Y 495.365,Z 522.726,A -85,B 0,C 180,E1 -6194.743,E2 -6194.743} C_VEL
LIN {X 0,Y 495.326,Z 525.359,A -85,B 0,C 180,E1 -6195.518,E2 -6195.518} C_VEL
LIN {X 0,Y 497.058,Z 538.145,A -85,B 0,C 180,E1 -6195.883,E2 -6195.883} C_VEL
LIN {X 0,Y 497.525,Z 542.874,A -85,B 0,C 180,E1 -6196.053,E2 -6196.053} C_VEL
LIN {X 0,Y 497.175,Z 556.269,A -85,B 0,C 180,E1 -6196.616,E2 -6196.616} C_VEL
LIN {X 0,Y 496.854,Z 568.235,A -85,B 0,C 180,E1 -6197.297,E2 -6197.297} C_VEL
LIN {X 0,Y 496.418,Z 580.066,A -85,B 0,C 180,E1 -6198.154,E2 -6198.154} C_VEL
LIN {X 0,Y 496.061,Z 590.236,A -85,B 0,C 180,E1 -6199.077,E2 -6199.077} C_VEL
LIN {X 0,Y 495.698,Z 600.279,A -85,B 0,C 180,E1 -6200.204,E2 -6200.204} C_VEL
LIN {X 0,Y 495.472,Z 609.139,A -85,B 0,C 180,E1 -6201.435,E2 -6201.435} C_VEL
LIN {X 0,Y 495.271,Z 616.195,A -85,B 0,C 180,E1 -6202.662,E2 -6202.662} C_VEL
LIN {X 0,Y 495.143,Z 622.385,A -85,B 0,C 180,E1 -6204.022,E2 -6204.022} C_VEL
LIN {X 0,Y 495.039,Z 626.288,A -85,B 0,C 180,E1 -6205.113,E2 -6205.113} C_VEL
LIN {X 0,Y 495.064,Z 628.641,A -85,B 0,C 180,E1 -6205.93,E2 -6205.93} C_VEL
LIN {X 0,Y 495.044,Z 630.554,A -85,B 0,C 180,E1 -6206.745,E2 -6206.745} C_VEL
LIN {X 0,Y 495.053,Z 631.986,A -85,B 0,C 180,E1 -6207.559,E2 -6207.559} C_VEL
LIN {X 0,Y 494.91,Z 633.63,A -85,B 0,C 180,E1 -6209.186,E2 -6209.186} C_VEL
LIN {X 0,Y 494.898,Z 633.862,A -85,B 0,C 180,E1 -6210,E2 -6210} C_VEL
LIN {X 0,Y 494.963,Z 633.045,A -85,B 0,C 180,E1 -6211.627,E2 -6211.627} C_VEL
LIN {X 0,Y 495.053,Z 632.05,A -85,B 0,C 180,E1 -6212.441,E2 -6212.441} C_VEL
LIN {X 0,Y 495.044,Z 630.639,A -85,B 0,C 180,E1 -6213.255,E2 -6213.255} C_VEL
LIN {X 0,Y 495.027,Z 627.671,A -85,B 0,C 180,E1 -6214.478,E2 -6214.478} C_VEL
LIN {X 0,Y 495.153,Z 623.655,A -85,B 0,C 180,E1 -6215.702,E2 -6215.702} C_VEL
LIN {X 0,Y 495.257,Z 617.461,A -85,B 0,C 180,E1 -6217.133,E2 -6217.133} C_VEL
LIN {X 0,Y 495.443,Z 610.701,A -85,B 0,C 180,E1 -6218.36,E2 -6218.36} C_VEL
LIN {X 0,Y 495.689,Z 602.318,A -85,B 0,C 180,E1 -6219.59,E2 -6219.59} C_VEL
LIN {X 0,Y 496.004,Z 593.7,A -85,B 0,C 180,E1 -6220.614,E2 -6220.614} C_VEL
LIN {X 0,Y 496.353,Z 583.08,A -85,B 0,C 180,E1 -6221.64,E2 -6221.64} C_VEL
LIN {X 0,Y 496.779,Z 571.522,A -85,B 0,C 180,E1 -6222.537,E2 -6222.537} C_VEL
LIN {X 0,Y 497.12,Z 561.092,A -85,B 0,C 180,E1 -6223.177,E2 -6223.177} C_VEL
LIN {X 0,Y 497.491,Z 549.23,A -85,B 0,C 180,E1 -6223.739,E2 -6223.739} C_VEL
LIN {X 0,Y 497.469,Z 540.551,A -85,B 0,C 180,E1 -6224.066,E2 -6224.066} C_VEL
LIN {X 0,Y 495.536,Z 527.657,A -85,B 0,C 180,E1 -6224.456,E2 -6224.456} C_VEL
LIN {X 0,Y 495.357,Z 526.037,A -85,B 0,C 180,E1 -6224.507,E2 -6224.507} C_VEL
LIN {X 0,Y 495.477,Z 517.181,A -85,B 0,C 180,E1 -6227.33,E2 -6227.33} C_VEL
LIN {X 0,Y 495.665,Z 508.103,A -85,B 0,C 180,E1 -6230.267,E2 -6230.267} C_VEL
LIN {X 0,Y 495.899,Z 498.653,A -85,B 0,C 180,E1 -6233.38,E2 -6233.38} C_VEL
LIN {X 0,Y 496.209,Z 489.619,A -85,B 0,C 180,E1 -6236.447,E2 -6236.447} C_VEL
LIN {X 0,Y 496.493,Z 481.655,A -85,B 0,C 180,E1 -6239.233,E2 -6239.233} C_VEL
LIN {X 0,Y 496.856,Z 474.153,A -85,B 0,C 180,E1 -6241.93,E2 -6241.93} C_VEL
LIN {X 0,Y 497.193,Z 466.079,A -85,B 0,C 180,E1 -6244.93,E2 -6244.93} C_VEL
LIN {X 0,Y 497.08,Z 462.235,A -85,B 0,C 180,E1 -6246.429,E2 -6246.429} C_VEL
LIN {X 0,Y 495.776,Z 454.732,A -85,B 0,C 180,E1 -6249.553,E2 -6249.553} C_VEL
LIN {X 0,Y 495.739,Z 454.735,A -85,B 0,C 180,E1 -6252.507,E2 -6252.507} C_VEL
LIN {X 0,Y 495.751,Z 454.732,A -85,B 0,C 180,E1 -6255.139,E2 -6255.139} C_VEL
LIN {X 0,Y 495.779,Z 454.729,A -85,B 0,C 180,E1 -6258.221,E2 -6258.221} C_VEL
LIN {X 0,Y 495.751,Z 454.73,A -85,B 0,C 180,E1 -6261.408,E2 -6261.408} C_VEL
LIN {X 0,Y 495.75,Z 454.733,A -85,B 0,C 180,E1 -6264.462,E2 -6264.462} C_VEL
LIN {X 0,Y 495.769,Z 454.729,A -85,B 0,C 180,E1 -6267.406,E2 -6267.406} C_VEL
LIN {X 0,Y 495.768,Z 454.733,A -85,B 0,C 180,E1 -6270.254,E2 -6270.254} C_VEL
LIN {X 0,Y 495.825,Z 454.725,A -85,B 0,C 180,E1 -6273.251,E2 -6273.251} C_VEL
LIN {X 0,Y 495.744,Z 454.731,A -85,B 0,C 180,E1 -6275.725,E2 -6275.725} C_VEL
LIN {X 0,Y 495.745,Z 454.734,A -85,B 0,C 180,E1 -6278.371,E2 -6278.371} C_VEL
LIN {X 0,Y 495.787,Z 454.731,A -85,B 0,C 180,E1 -6280.972,E2 -6280.972} C_VEL
LIN {X 0,Y 495.782,Z 454.727,A -85,B 0,C 180,E1 -6283.53,E2 -6283.53} C_VEL
LIN {X 0,Y 495.796,Z 454.728,A -85,B 0,C 180,E1 -6286.056,E2 -6286.056} C_VEL
LIN {X 0,Y 495.854,Z 454.721,A -85,B 0,C 180,E1 -6288.555,E2 -6288.555} C_VEL
LIN {X 0,Y 495.875,Z 454.718,A -85,B 0,C 180,E1 -6291.852,E2 -6291.852} C_VEL
LIN {X 0,Y 495.898,Z 454.714,A -85,B 0,C 180,E1 -6294.307,E2 -6294.307} C_VEL
LIN {X 0,Y 495.995,Z 454.7,A -85,B 0,C 180,E1 -6297.564,E2 -6297.564} C_VEL
LIN {X 0,Y 496.002,Z 454.704,A -85,B 0,C 180,E1 -6300,E2 -6300} C_VEL
LIN {X 0,Y 495.995,Z 454.702,A -85,B 0,C 180,E1 -6302.436,E2 -6302.436} C_VEL
LIN {X 0,Y 495.898,Z 454.714,A -85,B 0,C 180,E1 -6305.694,E2 -6305.694} C_VEL
LIN {X 0,Y 495.876,Z 454.717,A -85,B 0,C 180,E1 -6308.148,E2 -6308.148} C_VEL
LIN {X 0,Y 495.854,Z 454.717,A -85,B 0,C 180,E1 -6311.445,E2 -6311.445} C_VEL
LIN {X 0,Y 495.793,Z 454.727,A -85,B 0,C 180,E1 -6314.783,E2 -6314.783} C_VEL
LIN {X 0,Y 495.789,Z 454.727,A -85,B 0,C 180,E1 -6317.319,E2 -6317.319} C_VEL
LIN {X 0,Y 495.781,Z 454.729,A -85,B 0,C 180,E1 -6319.89,E2 -6319.89} C_VEL
LIN {X 0,Y 495.763,Z 454.733,A -85,B 0,C 180,E1 -6322.861,E2 -6322.861} C_VEL
LIN {X 0,Y 495.794,Z 454.728,A -85,B 0,C 180,E1 -6326.068,E2 -6326.068} C_VEL
LIN {X 0,Y 495.775,Z 454.729,A -85,B 0,C 180,E1 -6328.815,E2 -6328.815} C_VEL
LIN {X 0,Y 495.759,Z 454.73,A -85,B 0,C 180,E1 -6331.726,E2 -6331.726} C_VEL
LIN {X 0,Y 495.778,Z 454.728,A -85,B 0,C 180,E1 -6334.695,E2 -6334.695} C_VEL
LIN {X 0,Y 495.734,Z 454.736,A -85,B 0,C 180,E1 -6337.562,E2 -6337.562} C_VEL
LIN {X 0,Y 495.77,Z 454.729,A -85,B 0,C 180,E1 -6340.7,E2 -6340.7} C_VEL
LIN {X 0,Y 495.738,Z 454.736,A -85,B 0,C 180,E1 -6343.696,E2 -6343.696} C_VEL
LIN {X 0,Y 495.733,Z 454.736,A -85,B 0,C 180,E1 -6346.305,E2 -6346.305} C_VEL
LIN {X 0,Y 495.769,Z 454.73,A -85,B 0,C 180,E1 -6349.3,E2 -6349.3} C_VEL
LIN {X 0,Y 495.735,Z 454.736,A -85,B 0,C 180,E1 -6352.439,E2 -6352.439} C_VEL
LIN {X 0,Y 495.788,Z 454.726,A -85,B 0,C 180,E1 -6355.458,E2 -6355.458} C_VEL
LIN {X 0,Y 495.759,Z 454.731,A -85,B 0,C 180,E1 -6358.364,E2 -6358.364} C_VEL
LIN {X 0,Y 495.757,Z 454.729,A -85,B 0,C 180,E1 -6360.757,E2 -6360.757} C_VEL
LIN {X 0,Y 495.099,Z 454.812,A -85,B 0,C 180,E1 -6361.436,E2 -6361.436} C_VEL
LIN {X 0,Y 492.243,Z 455.169,A -85,B 0,C 180,E1 -6362.539,E2 -6362.539} C_VEL
LIN {X 0,Y 489.835,Z 455.469,A -85,B 0,C 180,E1 -6363.427,E2 -6363.427} C_VEL
LIN {X 0,Y 488.819,Z 455.597,A -85,B 0,C 180,E1 -6364.114,E2 -6364.114} C_VEL
LIN {X 0,Y 488.747,Z 455.604,A -85,B 0,C 180,E1 -6364.346,E2 -6364.346} C_VEL
LIN {X 0,Y 488.727,Z 455.608,A -85,B 0,C 180,E1 -6367.153,E2 -6367.153} C_VEL
LIN {X 0,Y 488.73,Z 455.608,A -85,B 0,C 180,E1 -6369.811,E2 -6369.811} C_VEL
LIN {X 0,Y 488.72,Z 455.608,A -85,B 0,C 180,E1 -6372.423,E2 -6372.423} C_VEL
LIN {X 0,Y 488.767,Z 455.602,A -85,B 0,C 180,E1 -6375,E2 -6375} C_VEL
LIN {X 0,Y 488.811,Z 455.596,A -85,B 0,C 180,E1 -6378.388,E2 -6378.388} C_VEL
LIN {X 0,Y 488.822,Z 455.595,A -85,B 0,C 180,E1 -6381.734,E2 -6381.734} C_VEL
LIN {X 0,Y 488.811,Z 455.596,A -85,B 0,C 180,E1 -6385.051,E2 -6385.051} C_VEL
LIN {X 0,Y 488.966,Z 455.579,A -85,B 0,C 180,E1 -6387.529,E2 -6387.529} C_VEL
LIN {X 0,Y 488.975,Z 455.578,A -85,B 0,C 180,E1 -6390,E2 -6390} C_VEL
LIN {X 0,Y 488.966,Z 455.576,A -85,B 0,C 180,E1 -6392.471,E2 -6392.471} C_VEL
LIN {X 0,Y 488.86,Z 455.59,A -85,B 0,C 180,E1 -6395.776,E2 -6395.776} C_VEL
LIN {X 0,Y 488.791,Z 455.6,A -85,B 0,C 180,E1 -6398.267,E2 -6398.267} C_VEL
LIN {X 0,Y 488.811,Z 455.598,A -85,B 0,C 180,E1 -6401.612,E2 -6401.612} C_VEL
LIN {X 0,Y 488.767,Z 455.6,A -85,B 0,C 180,E1 -6405,E2 -6405} C_VEL
LIN {X 0,Y 488.76,Z 455.603,A -85,B 0,C 180,E1 -6408.442,E2 -6408.442} C_VEL
LIN {X 0,Y 488.712,Z 455.609,A -85,B 0,C 180,E1 -6411.071,E2 -6411.071} C_VEL
LIN {X 0,Y 488.695,Z 455.614,A -85,B 0,C 180,E1 -6413.746,E2 -6413.746} C_VEL
LIN {X 0,Y 488.797,Z 455.6,A -85,B 0,C 180,E1 -6416.944,E2 -6416.944} C_VEL
LIN {X 0,Y 488.714,Z 455.608,A -85,B 0,C 180,E1 -6420.363,E2 -6420.363} C_VEL
LIN {X 0,Y 488.739,Z 455.606,A -85,B 0,C 180,E1 -6423.484,E2 -6423.484} C_VEL
LIN {X 0,Y 488.687,Z 455.612,A -85,B 0,C 180,E1 -6426.354,E2 -6426.354} C_VEL
LIN {X 0,Y 488.706,Z 455.612,A -85,B 0,C 180,E1 -6429.254,E2 -6429.254} C_VEL
LIN {X 0,Y 488.712,Z 455.609,A -85,B 0,C 180,E1 -6431.6,E2 -6431.6} C_VEL
LIN {X 0,Y 488.705,Z 455.607,A -85,B 0,C 180,E1 -6434.803,E2 -6434.803} C_VEL
LIN {X 0,Y 488.696,Z 455.612,A -85,B 0,C 180,E1 -6437.474,E2 -6437.474} C_VEL
LIN {X 0,Y 488.737,Z 455.606,A -85,B 0,C 180,E1 -6439.677,E2 -6439.677} C_VEL
LIN {X 0,Y 488.67,Z 455.614,A -85,B 0,C 180,E1 -6442.84,E2 -6442.84} C_VEL
LIN {X 0,Y 488.521,Z 455.636,A -85,B 0,C 180,E1 -6445.87,E2 -6445.87} C_VEL
LIN {X 0,Y 488.188,Z 455.723,A -85,B 0,C 180,E1 -6448.784,E2 -6448.784} C_VEL
LIN {X 0,Y 488.169,Z 458.723,A -85,B 0,C 180,E1 -6451.634,E2 -6451.634} C_VEL
LIN {X 0,Y 488.138,Z 461.702,A -85,B 0,C 180,E1 -6454.41,E2 -6454.41} C_VEL
LIN {X 0,Y 488.08,Z 464.667,A -85,B 0,C 180,E1 -6457.155,E2 -6457.155} C_VEL
LIN {X 0,Y 488.039,Z 467.542,A -85,B 0,C 180,E1 -6459.781,E2 -6459.781} C_VEL
LIN {X 0,Y 488.007,Z 470.443,A -85,B 0,C 180,E1 -6462.396,E2 -6462.396} C_VEL
LIN {X 0,Y 488.005,Z 473.932,A -85,B 0,C 180,E1 -6465.422,E2 -6465.422} C_VEL
LIN {X 0,Y 490.46,Z 485.938,A -85,B 0,C 180,E1 -6465.848,E2 -6465.848} C_VEL
LIN {X 0,Y 490.726,Z 490.182,A -85,B 0,C 180,E1 -6466.014,E2 -6466.014} C_VEL
LIN {X 0,Y 490.443,Z 501.599,A -85,B 0,C 180,E1 -6466.534,E2 -6466.534} C_VEL
LIN {X 0,Y 490.048,Z 513.735,A -85,B 0,C 180,E1 -6467.26,E2 -6467.26} C_VEL
LIN {X 0,Y 489.709,Z 524.688,A -85,B 0,C 180,E1 -6468.094,E2 -6468.094} C_VEL
LIN {X 0,Y 489.339,Z 534.556,A -85,B 0,C 180,E1 -6469.03,E2 -6469.03} C_VEL
LIN {X 0,Y 488.947,Z 543.535,A -85,B 0,C 180,E1 -6470.067,E2 -6470.067} C_VEL
LIN {X 0,Y 488.632,Z 552.308,A -85,B 0,C 180,E1 -6471.314,E2 -6471.314} C_VEL
LIN {X 0,Y 488.356,Z 559.308,A -85,B 0,C 180,E1 -6472.558,E2 -6472.558} C_VEL
LIN {X 0,Y 488.232,Z 565.34,A -85,B 0,C 180,E1 -6473.916,E2 -6473.916} C_VEL
LIN {X 0,Y 488.07,Z 570.545,A -85,B 0,C 180,E1 -6475.457,E2 -6475.457} C_VEL
LIN {X 0,Y 487.98,Z 573.528,A -85,B 0,C 180,E1 -6476.697,E2 -6476.697} C_VEL
LIN {X 0,Y 487.989,Z 574.964,A -85,B 0,C 180,E1 -6477.524,E2 -6477.524} C_VEL
LIN {X 0,Y 487.834,Z 576.635,A -85,B 0,C 180,E1 -6479.174,E2 -6479.174} C_VEL
LIN {X 0,Y 487.82,Z 576.895,A -85,B 0,C 180,E1 -6480,E2 -6480} C_VEL
LIN {X 0,Y 487.834,Z 576.72,A -85,B 0,C 180,E1 -6480.825,E2 -6480.825} C_VEL
LIN {X 0,Y 487.99,Z 575.186,A -85,B 0,C 180,E1 -6482.476,E2 -6482.476} C_VEL
LIN {X 0,Y 487.99,Z 573.837,A -85,B 0,C 180,E1 -6483.302,E2 -6483.302} C_VEL
LIN {X 0,Y 488.073,Z 570.97,A -85,B 0,C 180,E1 -6484.542,E2 -6484.542} C_VEL
LIN {X 0,Y 488.181,Z 567.07,A -85,B 0,C 180,E1 -6485.784,E2 -6485.784} C_VEL
LIN {X 0,Y 488.335,Z 561.134,A -85,B 0,C 180,E1 -6487.213,E2 -6487.213} C_VEL
LIN {X 0,Y 488.579,Z 554.418,A -85,B 0,C 180,E1 -6488.479,E2 -6488.479} C_VEL
LIN {X 0,Y 488.867,Z 546.192,A -85,B 0,C 180,E1 -6489.725,E2 -6489.725} C_VEL
LIN {X 0,Y 489.177,Z 537.711,A -85,B 0,C 180,E1 -6490.764,E2 -6490.764} C_VEL
LIN {X 0,Y 489.704,Z 527.245,A -85,B 0,C 180,E1 -6491.801,E2 -6491.801} C_VEL
LIN {X 0,Y 490.015,Z 516.403,A -85,B 0,C 180,E1 -6492.671,E2 -6492.671} C_VEL
LIN {X 0,Y 490.384,Z 505.55,A -85,B 0,C 180,E1 -6493.362,E2 -6493.362} C_VEL
LIN {X 0,Y 490.74,Z 492.7,A -85,B 0,C 180,E1 -6493.985,E2 -6493.985} C_VEL
LIN {X 0,Y 490.573,Z 486.589,A -85,B 0,C 180,E1 -6494.228,E2 -6494.228} C_VEL
LIN {X 0,Y 488.588,Z 477.171,A -85,B 0,C 180,E1 -6494.58,E2 -6494.58} C_VEL
LIN {X 0,Y 488.126,Z 475.11,A -85,B 0,C 180,E1 -6494.674,E2 -6494.674} C_VEL
LIN {X 0,Y 488.158,Z 472.186,A -85,B 0,C 180,E1 -6497.598,E2 -6497.598} C_VEL
LIN {X 0,Y 488.229,Z 468.822,A -85,B 0,C 180,E1 -6501.092,E2 -6501.092} C_VEL
LIN {X 0,Y 488.316,Z 466.353,A -85,B 0,C 180,E1 -6503.765,E2 -6503.765} C_VEL
LIN {X 0,Y 488.474,Z 463.627,A -85,B 0,C 180,E1 -6506.869,E2 -6506.869} C_VEL
LIN {X 0,Y 488.561,Z 461.647,A -85,B 0,C 180,E1 -6509.281,E2 -6509.281} C_VEL
LIN {X 0,Y 488.71,Z 459.432,A -85,B 0,C 180,E1 -6512.147,E2 -6512.147} C_VEL
LIN {X 0,Y 488.828,Z 457.436,A -85,B 0,C 180,E1 -6515.106,E2 -6515.106} C_VEL
LIN {X 0,Y 488.743,Z 456.058,A -85,B 0,C 180,E1 -6517.731,E2 -6517.731} C_VEL
LIN {X 0,Y 488.704,Z 455.614,A -85,B 0,C 180,E1 -6519.254,E2 -6519.254} C_VEL
LIN {X 0,Y 488.726,Z 455.61,A -85,B 0,C 180,E1 -6521.602,E2 -6521.602} C_VEL
LIN {X 0,Y 488.715,Z 455.612,A -85,B 0,C 180,E1 -6524.801,E2 -6524.801} C_VEL
LIN {X 0,Y 488.773,Z 456.157,A -85,B 0,C 180,E1 -6526.355,E2 -6526.355} C_VEL
LIN {X 0,Y 489.166,Z 457.949,A -85,B 0,C 180,E1 -6528.631,E2 -6528.631} C_VEL
LIN {X 0,Y 489.615,Z 460.526,A -85,B 0,C 180,E1 -6530.833,E2 -6530.833} C_VEL
LIN {X 0,Y 490.22,Z 464.518,A -85,B 0,C 180,E1 -6533.402,E2 -6533.402} C_VEL
LIN {X 0,Y 490.249,Z 467.629,A -85,B 0,C 180,E1 -6535.011,E2 -6535.011} C_VEL
LIN {X 0,Y 489.759,Z 472.985,A -85,B 0,C 180,E1 -6537.444,E2 -6537.444} C_VEL
LIN {X 0,Y 489.314,Z 480,A -85,B 0,C 180,E1 -6540.296,E2 -6540.296} C_VEL
LIN {X 0,Y 489.05,Z 487.26,A -85,B 0,C 180,E1 -6542.998,E2 -6542.998} C_VEL
LIN {X 0,Y 488.757,Z 495.298,A -85,B 0,C 180,E1 -6545.807,E2 -6545.807} C_VEL
LIN {X 0,Y 488.553,Z 504.65,A -85,B 0,C 180,E1 -6548.922,E2 -6548.922} C_VEL
LIN {X 0,Y 488.349,Z 514.488,A -85,B 0,C 180,E1 -6552.085,E2 -6552.085} C_VEL
LIN {X 0,Y 488.26,Z 524.398,A -85,B 0,C 180,E1 -6555.197,E2 -6555.197} C_VEL
LIN {X 0,Y 488.24,Z 524.739,A -85,B 0,C 180,E1 -6555.303,E2 -6555.303} C_VEL
LIN {X 0,Y 490.053,Z 538.613,A -85,B 0,C 180,E1 -6555.717,E2 -6555.717} C_VEL
LIN {X 0,Y 490.577,Z 543.536,A -85,B 0,C 180,E1 -6555.904,E2 -6555.904} C_VEL
LIN {X 0,Y 490.236,Z 555.529,A -85,B 0,C 180,E1 -6556.423,E2 -6556.423} C_VEL
LIN {X 0,Y 489.871,Z 566.988,A -85,B 0,C 180,E1 -6557.078,E2 -6557.078} C_VEL
LIN {X 0,Y 489.441,Z 579.396,A -85,B 0,C 180,E1 -6557.982,E2 -6557.982} C_VEL
LIN {X 0,Y 489.065,Z 589.62,A -85,B 0,C 180,E1 -6558.919,E2 -6558.919} C_VEL
LIN {X 0,Y 488.65,Z 599.697,A -85,B 0,C 180,E1 -6560.061,E2 -6560.061} C_VEL
LIN {X 0,Y 488.387,Z 608.594,A -85,B 0,C 180,E1 -6561.309,E2 -6561.309} C_VEL
LIN {X 0,Y 488.194,Z 615.684,A -85,B 0,C 180,E1 -6562.556,E2 -6562.556} C_VEL
LIN {X 0,Y 488.038,Z 621.27,A -85,B 0,C 180,E1 -6563.776,E2 -6563.776} C_VEL
LIN {X 0,Y 487.97,Z 625.826,A -85,B 0,C 180,E1 -6565.042,E2 -6565.042} C_VEL
LIN {X 0,Y 487.962,Z 628.193,A -85,B 0,C 180,E1 -6565.87,E2 -6565.87} C_VEL
LIN {X 0,Y 487.969,Z 630.118,A -85,B 0,C 180,E1 -6566.697,E2 -6566.697} C_VEL
LIN {X 0,Y 487.972,Z 631.558,A -85,B 0,C 180,E1 -6567.524,E2 -6567.524} C_VEL
LIN {X 0,Y 487.834,Z 633.218,A -85,B 0,C 180,E1 -6569.174,E2 -6569.174} C_VEL
LIN {X 0,Y 487.819,Z 633.453,A -85,B 0,C 180,E1 -6570,E2 -6570} C_VEL
LIN {X 0,Y 487.893,Z 632.64,A -85,B 0,C 180,E1 -6571.651,E2 -6571.651} C_VEL
LIN {X 0,Y 487.959,Z 631.645,A -85,B 0,C 180,E1 -6572.476,E2 -6572.476} C_VEL
LIN {X 0,Y 487.968,Z 630.232,A -85,B 0,C 180,E1 -6573.303,E2 -6573.303} C_VEL
LIN {X 0,Y 487.936,Z 627.259,A -85,B 0,C 180,E1 -6574.544,E2 -6574.544} C_VEL
LIN {X 0,Y 488.049,Z 623.234,A -85,B 0,C 180,E1 -6575.785,E2 -6575.785} C_VEL
LIN {X 0,Y 488.182,Z 617.027,A -85,B 0,C 180,E1 -6577.237,E2 -6577.237} C_VEL
LIN {X 0,Y 488.372,Z 610.255,A -85,B 0,C 180,E1 -6578.482,E2 -6578.482} C_VEL
LIN {X 0,Y 488.628,Z 601.854,A -85,B 0,C 180,E1 -6579.73,E2 -6579.73} C_VEL
LIN {X 0,Y 488.991,Z 593.216,A -85,B 0,C 180,E1 -6580.768,E2 -6580.768} C_VEL
LIN {X 0,Y 489.373,Z 582.585,A -85,B 0,C 180,E1 -6581.809,E2 -6581.809} C_VEL
LIN {X 0,Y 489.763,Z 572.185,A -85,B 0,C 180,E1 -6582.633,E2 -6582.633} C_VEL
LIN {X 0,Y 490.16,Z 560.547,A -85,B 0,C 180,E1 -6583.368,E2 -6583.368} C_VEL
LIN {X 0,Y 490.56,Z 548.661,A -85,B 0,C 180,E1 -6583.937,E2 -6583.937} C_VEL
LIN {X 0,Y 490.494,Z 541.101,A -85,B 0,C 180,E1 -6584.23,E2 -6584.23} C_VEL
LIN {X 0,Y 488.552,Z 527.784,A -85,B 0,C 180,E1 -6584.654,E2 -6584.654} C_VEL
LIN {X 0,Y 488.29,Z 525.713,A -85,B 0,C 180,E1 -6584.722,E2 -6584.722} C_VEL
LIN {X 0,Y 488.437,Z 515.845,A -85,B 0,C 180,E1 -6587.933,E2 -6587.933} C_VEL
LIN {X 0,Y 488.654,Z 506.35,A -85,B 0,C 180,E1 -6591.073,E2 -6591.073} C_VEL
LIN {X 0,Y 488.942,Z 497.142,A -85,B 0,C 180,E1 -6594.183,E2 -6594.183} C_VEL
LIN {X 0,Y 489.299,Z 488.004,A -85,B 0,C 180,E1 -6597.363,E2 -6597.363} C_VEL
LIN {X 0,Y 489.662,Z 479.122,A -85,B 0,C 180,E1 -6600.552,E2 -6600.552} C_VEL
LIN {X 0,Y 489.998,Z 472.417,A -85,B 0,C 180,E1 -6603.027,E2 -6603.027} C_VEL
LIN {X 0,Y 490.306,Z 465.819,A -85,B 0,C 180,E1 -6605.55,E2 -6605.55} C_VEL
LIN {X 0,Y 489.879,Z 462.102,A -85,B 0,C 180,E1 -6607.053,E2 -6607.053} C_VEL
LIN {X 0,Y 488.732,Z 455.61,A -85,B 0,C 180,E1 -6609.852,E2 -6609.852} C_VEL
LIN {X 0,Y 488.711,Z 455.612,A -85,B 0,C 180,E1 -6612.826,E2 -6612.826} C_VEL
LIN {X 0,Y 488.704,Z 455.613,A -85,B 0,C 180,E1 -6615.976,E2 -6615.976} C_VEL
LIN {X 0,Y 488.72,Z 455.608,A -85,B 0,C 180,E1 -6618.586,E2 -6618.586} C_VEL
LIN {X 0,Y 488.681,Z 455.612,A -85,B 0,C 180,E1 -6621.8,E2 -6621.8} C_VEL
LIN {X 0,Y 488.725,Z 455.609,A -85,B 0,C 180,E1 -6625.052,E2 -6625.052} C_VEL
LIN {X 0,Y 488.705,Z 455.608,A -85,B 0,C 180,E1 -6628.046,E2 -6628.046} C_VEL
LIN {X 0,Y 488.725,Z 455.607,A -85,B 0,C 180,E1 -6630.73,E2 -6630.73} C_VEL
LIN {X 0,Y 488.758,Z 455.604,A -85,B 0,C 180,E1 -6633.528,E2 -6633.528} C_VEL
LIN {X 0,Y 488.686,Z 455.613,A -85,B 0,C 180,E1 -6636.254,E2 -6636.254} C_VEL
LIN {X 0,Y 488.748,Z 455.606,A -85,B 0,C 180,E1 -6639.176,E2 -6639.176} C_VEL
LIN {X 0,Y 488.761,Z 455.602,A -85,B 0,C 180,E1 -6641.628,E2 -6641.628} C_VEL
LIN {X 0,Y 488.764,Z 455.602,A -85,B 0,C 180,E1 -6645,E2 -6645} C_VEL
LIN {X 0,Y 488.808,Z 455.597,A -85,B 0,C 180,E1 -6648.388,E2 -6648.388} C_VEL
LIN {X 0,Y 488.819,Z 455.596,A -85,B 0,C 180,E1 -6651.734,E2 -6651.734} C_VEL
LIN {X 0,Y 488.857,Z 455.591,A -85,B 0,C 180,E1 -6654.224,E2 -6654.224} C_VEL
LIN {X 0,Y 488.963,Z 455.576,A -85,B 0,C 180,E1 -6657.529,E2 -6657.529} C_VEL
LIN {X 0,Y 488.958,Z 455.579,A -85,B 0,C 180,E1 -6660.824,E2 -6660.824} C_VEL
LIN {X 0,Y 488.963,Z 455.579,A -85,B 0,C 180,E1 -6662.472,E2 -6662.472} C_VEL
LIN {X 0,Y 488.857,Z 455.591,A -85,B 0,C 180,E1 -6665.776,E2 -6665.776} C_VEL
LIN {X 0,Y 488.82,Z 455.595,A -85,B 0,C 180,E1 -6668.267,E2 -6668.267} C_VEL
LIN {X 0,Y 488.808,Z 455.595,A -85,B 0,C 180,E1 -6671.613,E2 -6671.613} C_VEL
LIN {X 0,Y 488.765,Z 455.604,A -85,B 0,C 180,E1 -6675.001,E2 -6675.001} C_VEL
LIN {X 0,Y 488.758,Z 455.607,A -85,B 0,C 180,E1 -6678.442,E2 -6678.442} C_VEL
LIN {X 0,Y 488.71,Z 455.609,A -85,B 0,C 180,E1 -6681.071,E2 -6681.071} C_VEL
LIN {X 0,Y 488.692,Z 455.611,A -85,B 0,C 180,E1 -6683.746,E2 -6683.746} C_VEL
LIN {X 0,Y 488.795,Z 455.597,A -85,B 0,C 180,E1 -6686.944,E2 -6686.944} C_VEL
LIN {X 0,Y 488.713,Z 455.609,A -85,B 0,C 180,E1 -6690.363,E2 -6690.363} C_VEL
LIN {X 0,Y 488.739,Z 455.603,A -85,B 0,C 180,E1 -6693.485,E2 -6693.485} C_VEL
LIN {X 0,Y 488.692,Z 455.611,A -85,B 0,C 180,E1 -6696.356,E2 -6696.356} C_VEL
LIN {X 0,Y 488.704,Z 455.609,A -85,B 0,C 180,E1 -6699.254,E2 -6699.254} C_VEL
LIN {X 0,Y 488.727,Z 455.607,A -85,B 0,C 180,E1 -6701.602,E2 -6701.602} C_VEL
LIN {X 0,Y 488.716,Z 455.611,A -85,B 0,C 180,E1 -6704.802,E2 -6704.802} C_VEL
LIN {X 0,Y 488.695,Z 455.609,A -85,B 0,C 180,E1 -6707.475,E2 -6707.475} C_VEL
LIN {X 0,Y 488.736,Z 455.608,A -85,B 0,C 180,E1 -6709.677,E2 -6709.677} C_VEL
LIN {X 0,Y 488.686,Z 455.614,A -85,B 0,C 180,E1 -6712.842,E2 -6712.842} C_VEL
LIN {X 0,Y 488.738,Z 455.608,A -85,B 0,C 180,E1 -6715.888,E2 -6715.888} C_VEL
LIN {X 0,Y 488.696,Z 455.613,A -85,B 0,C 180,E1 -6718.821,E2 -6718.821} C_VEL
LIN {X 0,Y 488.748,Z 455.604,A -85,B 0,C 180,E1 -6721.671,E2 -6721.671} C_VEL
LIN {X 0,Y 488.747,Z 455.604,A -85,B 0,C 180,E1 -6724.346,E2 -6724.346} C_VEL
LIN {X 0,Y 488.102,Z 455.687,A -85,B 0,C 180,E1 -6725.034,E2 -6725.034} C_VEL
LIN {X 0,Y 485.233,Z 456.045,A -85,B 0,C 180,E1 -6726.15,E2 -6726.15} C_VEL
LIN {X 0,Y 482.787,Z 456.348,A -85,B 0,C 180,E1 -6727.05,E2 -6727.05} C_VEL
LIN {X 0,Y 481.729,Z 456.478,A -85,B 0,C 180,E1 -6727.745,E2 -6727.745} C_VEL
LIN {X 0,Y 481.64,Z 456.488,A -85,B 0,C 180,E1 -6727.981,E2 -6727.981} C_VEL
LIN {X 0,Y 481.709,Z 456.481,A -85,B 0,C 180,E1 -6730.393,E2 -6730.393} C_VEL
LIN {X 0,Y 481.684,Z 456.486,A -85,B 0,C 180,E1 -6733.034,E2 -6733.034} C_VEL
LIN {X 0,Y 481.695,Z 456.482,A -85,B 0,C 180,E1 -6735.639,E2 -6735.639} C_VEL
LIN {X 0,Y 481.756,Z 456.476,A -85,B 0,C 180,E1 -6738.215,E2 -6738.215} C_VEL
LIN {X 0,Y 481.767,Z 456.474,A -85,B 0,C 180,E1 -6741.612,E2 -6741.612} C_VEL
LIN {X 0,Y 481.781,Z 456.471,A -85,B 0,C 180,E1 -6744.979,E2 -6744.979} C_VEL
LIN {X 0,Y 481.933,Z 456.455,A -85,B 0,C 180,E1 -6747.493,E2 -6747.493} C_VEL
LIN {X 0,Y 481.946,Z 456.454,A -85,B 0,C 180,E1 -6750,E2 -6750} C_VEL
LIN {X 0,Y 481.933,Z 456.453,A -85,B 0,C 180,E1 -6752.508,E2 -6752.508} C_VEL
LIN {X 0,Y 481.821,Z 456.467,A -85,B 0,C 180,E1 -6755.86,E2 -6755.86} C_VEL
LIN {X 0,Y 481.746,Z 456.476,A -85,B 0,C 180,E1 -6758.389,E2 -6758.389} C_VEL
LIN {X 0,Y 481.756,Z 456.476,A -85,B 0,C 180,E1 -6761.785,E2 -6761.785} C_VEL
LIN {X 0,Y 481.748,Z 456.475,A -85,B 0,C 180,E1 -6765.224,E2 -6765.224} C_VEL
LIN {X 0,Y 481.717,Z 456.482,A -85,B 0,C 180,E1 -6768.722,E2 -6768.722} C_VEL
LIN {X 0,Y 481.651,Z 456.488,A -85,B 0,C 180,E1 -6771.395,E2 -6771.395} C_VEL
LIN {X 0,Y 481.68,Z 456.485,A -85,B 0,C 180,E1 -6774.113,E2 -6774.113} C_VEL
LIN {X 0,Y 481.752,Z 456.477,A -85,B 0,C 180,E1 -6777.139,E2 -6777.139} C_VEL
LIN {X 0,Y 481.684,Z 456.487,A -85,B 0,C 180,E1 -6779.741,E2 -6779.741} C_VEL
LIN {X 0,Y 481.677,Z 456.486,A -85,B 0,C 180,E1 -6782.674,E2 -6782.674} C_VEL
LIN {X 0,Y 481.641,Z 456.49,A -85,B 0,C 180,E1 -6785.709,E2 -6785.709} C_VEL
LIN {X 0,Y 481.676,Z 456.485,A -85,B 0,C 180,E1 -6788.859,E2 -6788.859} C_VEL
LIN {X 0,Y 481.657,Z 456.489,A -85,B 0,C 180,E1 -6791.913,E2 -6791.913} C_VEL
LIN {X 0,Y 481.659,Z 456.486,A -85,B 0,C 180,E1 -6794.458,E2 -6794.458} C_VEL
LIN {X 0,Y 481.652,Z 456.488,A -85,B 0,C 180,E1 -6797.839,E2 -6797.839} C_VEL
LIN {X 0,Y 481.684,Z 456.484,A -85,B 0,C 180,E1 -6800.651,E2 -6800.651} C_VEL
LIN {X 0,Y 481.618,Z 456.496,A -85,B 0,C 180,E1 -6803.378,E2 -6803.378} C_VEL
LIN {X 0,Y 481.424,Z 456.519,A -85,B 0,C 180,E1 -6806.307,E2 -6806.307} C_VEL
LIN {X 0,Y 481.192,Z 456.549,A -85,B 0,C 180,E1 -6808.278,E2 -6808.278} C_VEL
LIN {X 0,Y 481.141,Z 457.142,A -85,B 0,C 180,E1 -6809.521,E2 -6809.521} C_VEL
LIN {X 0,Y 481.084,Z 459.901,A -85,B 0,C 180,E1 -6812.129,E2 -6812.129} C_VEL
LIN {X 0,Y 481.049,Z 462.883,A -85,B 0,C 180,E1 -6814.932,E2 -6814.932} C_VEL
LIN {X 0,Y 480.975,Z 465.85,A -85,B 0,C 180,E1 -6817.672,E2 -6817.672} C_VEL
LIN {X 0,Y 480.936,Z 468.777,A -85,B 0,C 180,E1 -6820.36,E2 -6820.36} C_VEL
LIN {X 0,Y 480.901,Z 471.708,A -85,B 0,C 180,E1 -6823.005,E2 -6823.005} C_VEL
LIN {X 0,Y 480.933,Z 474.169,A -85,B 0,C 180,E1 -6825.204,E2 -6825.204} C_VEL
LIN {X 0,Y 483.617,Z 487.05,A -85,B 0,C 180,E1 -6825.68,E2 -6825.68} C_VEL
LIN {X 0,Y 483.85,Z 491.6,A -85,B 0,C 180,E1 -6825.865,E2 -6825.865} C_VEL
LIN {X 0,Y 483.494,Z 503.709,A -85,B 0,C 180,E1 -6826.444,E2 -6826.444} C_VEL
LIN {X 0,Y 483.098,Z 515.215,A -85,B 0,C 180,E1 -6827.162,E2 -6827.162} C_VEL
LIN {X 0,Y 482.728,Z 526.091,A -85,B 0,C 180,E1 -6828.026,E2 -6828.026} C_VEL
LIN {X 0,Y 482.22,Z 536.761,A -85,B 0,C 180,E1 -6829.078,E2 -6829.078} C_VEL
LIN {X 0,Y 481.912,Z 545.442,A -85,B 0,C 180,E1 -6830.133,E2 -6830.133} C_VEL
LIN {X 0,Y 481.565,Z 553.869,A -85,B 0,C 180,E1 -6831.397,E2 -6831.397} C_VEL
LIN {X 0,Y 481.302,Z 560.647,A -85,B 0,C 180,E1 -6832.659,E2 -6832.659} C_VEL
LIN {X 0,Y 481.138,Z 566.87,A -85,B 0,C 180,E1 -6834.131,E2 -6834.131} C_VEL
LIN {X 0,Y 481.004,Z 570.917,A -85,B 0,C 180,E1 -6835.391,E2 -6835.391} C_VEL
LIN {X 0,Y 480.913,Z 573.914,A -85,B 0,C 180,E1 -6836.649,E2 -6836.649} C_VEL
LIN {X 0,Y 480.926,Z 575.359,A -85,B 0,C 180,E1 -6837.487,E2 -6837.487} C_VEL
LIN {X 0,Y 480.761,Z 577.044,A -85,B 0,C 180,E1 -6839.162,E2 -6839.162} C_VEL
LIN {X 0,Y 480.744,Z 577.307,A -85,B 0,C 180,E1 -6840,E2 -6840} C_VEL
LIN {X 0,Y 480.76,Z 577.134,A -85,B 0,C 180,E1 -6840.837,E2 -6840.837} C_VEL
LIN {X 0,Y 480.928,Z 575.601,A -85,B 0,C 180,E1 -6842.513,E2 -6842.513} C_VEL
LIN {X 0,Y 480.922,Z 574.25,A -85,B 0,C 180,E1 -6843.351,E2 -6843.351} C_VEL
LIN {X 0,Y 481.008,Z 571.379,A -85,B 0,C 180,E1 -6844.609,E2 -6844.609} C_VEL
LIN {X 0,Y 481.186,Z 566.446,A -85,B 0,C 180,E1 -6846.143,E2 -6846.143} C_VEL
LIN {X 0,Y 481.349,Z 560.415,A -85,B 0,C 180,E1 -6847.551,E2 -6847.551} C_VEL
LIN {X 0,Y 481.635,Z 553.555,A -85,B 0,C 180,E1 -6848.813,E2 -6848.813} C_VEL
LIN {X 0,Y 481.95,Z 544.942,A -85,B 0,C 180,E1 -6850.078,E2 -6850.078} C_VEL
LIN {X 0,Y 482.354,Z 536.116,A -85,B 0,C 180,E1 -6851.131,E2 -6851.131} C_VEL
LIN {X 0,Y 482.835,Z 526.424,A -85,B 0,C 180,E1 -6852.078,E2 -6852.078} C_VEL
LIN {X 0,Y 483.15,Z 515.53,A -85,B 0,C 180,E1 -6852.941,E2 -6852.941} C_VEL
LIN {X 0,Y 483.542,Z 503.954,A -85,B 0,C 180,E1 -6853.661,E2 -6853.661} C_VEL
LIN {X 0,Y 483.881,Z 491.82,A -85,B 0,C 180,E1 -6854.241,E2 -6854.241} C_VEL
LIN {X 0,Y 483.669,Z 487.322,A -85,B 0,C 180,E1 -6854.422,E2 -6854.422} C_VEL
LIN {X 0,Y 481.065,Z 475.672,A -85,B 0,C 180,E1 -6854.867,E2 -6854.867} C_VEL
LIN {X 0,Y 481.136,Z 472.3,A -85,B 0,C 180,E1 -6858.293,E2 -6858.293} C_VEL
LIN {X 0,Y 481.218,Z 469.915,A -85,B 0,C 180,E1 -6860.82,E2 -6860.82} C_VEL
LIN {X 0,Y 481.29,Z 466.926,A -85,B 0,C 180,E1 -6864.134,E2 -6864.134} C_VEL
LIN {X 0,Y 481.441,Z 464.437,A -85,B 0,C 180,E1 -6867.067,E2 -6867.067} C_VEL
LIN {X 0,Y 481.54,Z 462.297,A -85,B 0,C 180,E1 -6869.751,E2 -6869.751} C_VEL
LIN {X 0,Y 481.718,Z 460.159,A -85,B 0,C 180,E1 -6872.671,E2 -6872.671} C_VEL
LIN {X 0,Y 481.847,Z 458.558,A -85,B 0,C 180,E1 -6875.235,E2 -6875.235} C_VEL
LIN {X 0,Y 481.758,Z 457.246,A -85,B 0,C 180,E1 -6878.022,E2 -6878.022} C_VEL
LIN {X 0,Y 481.665,Z 456.49,A -85,B 0,C 180,E1 -6881.041,E2 -6881.041} C_VEL
LIN {X 0,Y 481.669,Z 456.551,A -85,B 0,C 180,E1 -6883.297,E2 -6883.297} C_VEL
LIN {X 0,Y 481.815,Z 457.307,A -85,B 0,C 180,E1 -6885.622,E2 -6885.622} C_VEL
LIN {X 0,Y 482.106,Z 458.989,A -85,B 0,C 180,E1 -6888.027,E2 -6888.027} C_VEL
LIN {X 0,Y 482.612,Z 461.652,A -85,B 0,C 180,E1 -6890.517,E2 -6890.517} C_VEL
LIN {X 0,Y 483.221,Z 465.517,A -85,B 0,C 180,E1 -6893.123,E2 -6893.123} C_VEL
LIN {X 0,Y 483.35,Z 468.049,A -85,B 0,C 180,E1 -6894.514,E2 -6894.514} C_VEL
LIN {X 0,Y 482.923,Z 473.067,A -85,B 0,C 180,E1 -6896.925,E2 -6896.925} C_VEL
LIN {X 0,Y 482.377,Z 479.931,A -85,B 0,C 180,E1 -6899.824,E2 -6899.824} C_VEL
LIN {X 0,Y 481.986,Z 488.574,A -85,B 0,C 180,E1 -6903.126,E2 -6903.126} C_VEL
LIN {X 0,Y 481.706,Z 496.333,A -85,B 0,C 180,E1 -6905.888,E2 -6905.888} C_VEL
LIN {X 0,Y 481.489,Z 505.761,A -85,B 0,C 180,E1 -6909.095,E2 -6909.095} C_VEL
LIN {X 0,Y 481.251,Z 515.062,A -85,B 0,C 180,E1 -6912.141,E2 -6912.141} C_VEL
LIN {X 0,Y 481.177,Z 524.244,A -85,B 0,C 180,E1 -6915.082,E2 -6915.082} C_VEL
LIN {X 0,Y 483.027,Z 538.704,A -85,B 0,C 180,E1 -6915.531,E2 -6915.531} C_VEL
LIN {X 0,Y 483.616,Z 544.224,A -85,B 0,C 180,E1 -6915.751,E2 -6915.751} C_VEL
LIN {X 0,Y 483.233,Z 556.789,A -85,B 0,C 180,E1 -6916.33,E2 -6916.33} C_VEL
LIN {X 0,Y 482.848,Z 568.989,A -85,B 0,C 180,E1 -6917.069,E2 -6917.069} C_VEL
LIN {X 0,Y 482.399,Z 580.026,A -85,B 0,C 180,E1 -6917.914,E2 -6917.914} C_VEL
LIN {X 0,Y 482.007,Z 589.992,A -85,B 0,C 180,E1 -6918.861,E2 -6918.861} C_VEL
LIN {X 0,Y 481.61,Z 599.115,A -85,B 0,C 180,E1 -6919.915,E2 -6919.915} C_VEL
LIN {X 0,Y 481.317,Z 608.049,A -85,B 0,C 180,E1 -6921.181,E2 -6921.181} C_VEL
LIN {X 0,Y 481.107,Z 615.172,A -85,B 0,C 180,E1 -6922.445,E2 -6922.445} C_VEL
LIN {X 0,Y 480.94,Z 621.276,A -85,B 0,C 180,E1 -6923.807,E2 -6923.807} C_VEL
LIN {X 0,Y 480.905,Z 625.368,A -85,B 0,C 180,E1 -6924.969,E2 -6924.969} C_VEL
LIN {X 0,Y 480.861,Z 627.745,A -85,B 0,C 180,E1 -6925.809,E2 -6925.809} C_VEL
LIN {X 0,Y 480.894,Z 629.681,A -85,B 0,C 180,E1 -6926.649,E2 -6926.649} C_VEL
LIN {X 0,Y 480.881,Z 631.129,A -85,B 0,C 180,E1 -6927.487,E2 -6927.487} C_VEL
LIN {X 0,Y 480.825,Z 632.165,A -85,B 0,C 180,E1 -6928.325,E2 -6928.325} C_VEL
LIN {X 0,Y 480.76,Z 632.806,A -85,B 0,C 180,E1 -6929.162,E2 -6929.162} C_VEL
LIN {X 0,Y 480.742,Z 633.044,A -85,B 0,C 180,E1 -6930,E2 -6930} C_VEL
LIN {X 0,Y 480.824,Z 632.237,A -85,B 0,C 180,E1 -6931.675,E2 -6931.675} C_VEL
LIN {X 0,Y 480.869,Z 631.24,A -85,B 0,C 180,E1 -6932.513,E2 -6932.513} C_VEL
LIN {X 0,Y 480.894,Z 629.825,A -85,B 0,C 180,E1 -6933.351,E2 -6933.351} C_VEL
LIN {X 0,Y 480.852,Z 626.846,A -85,B 0,C 180,E1 -6934.611,E2 -6934.611} C_VEL
LIN {X 0,Y 480.95,Z 622.813,A -85,B 0,C 180,E1 -6935.871,E2 -6935.871} C_VEL
LIN {X 0,Y 481.108,Z 616.593,A -85,B 0,C 180,E1 -6937.344,E2 -6937.344} C_VEL
LIN {X 0,Y 481.315,Z 609.808,A -85,B 0,C 180,E1 -6938.608,E2 -6938.608} C_VEL
LIN {X 0,Y 481.582,Z 601.39,A -85,B 0,C 180,E1 -6939.873,E2 -6939.873} C_VEL
LIN {X 0,Y 481.974,Z 592.731,A -85,B 0,C 180,E1 -6940.927,E2 -6940.927} C_VEL
LIN {X 0,Y 482.338,Z 582.086,A -85,B 0,C 180,E1 -6941.984,E2 -6941.984} C_VEL
LIN {X 0,Y 482.849,Z 570.561,A -85,B 0,C 180,E1 -6942.899,E2 -6942.899} C_VEL
LIN {X 0,Y 483.309,Z 558.036,A -85,B 0,C 180,E1 -6943.668,E2 -6943.668} C_VEL
LIN {X 0,Y 483.715,Z 545.615,A -85,B 0,C 180,E1 -6944.246,E2 -6944.246} C_VEL
LIN {X 0,Y 483.281,Z 539.802,A -85,B 0,C 180,E1 -6944.474,E2 -6944.474} C_VEL
LIN {X 0,Y 481.295,Z 526.442,A -85,B 0,C 180,E1 -6944.893,E2 -6944.893} C_VEL
LIN {X 0,Y 481.208,Z 525.475,A -85,B 0,C 180,E1 -6944.916,E2 -6944.916} C_VEL
LIN {X 0,Y 481.418,Z 514.99,A -85,B 0,C 180,E1 -6948.394,E2 -6948.394} C_VEL
LIN {X 0,Y 481.658,Z 504.779,A -85,B 0,C 180,E1 -6951.844,E2 -6951.844} C_VEL
LIN {X 0,Y 481.931,Z 496.935,A -85,B 0,C 180,E1 -6954.558,E2 -6954.558} C_VEL
LIN {X 0,Y 482.322,Z 487.818,A -85,B 0,C 180,E1 -6957.793,E2 -6957.793} C_VEL
LIN {X 0,Y 482.754,Z 478.643,A -85,B 0,C 180,E1 -6961.15,E2 -6961.15} C_VEL
LIN {X 0,Y 483.129,Z 471.17,A -85,B 0,C 180,E1 -6963.986,E2 -6963.986} C_VEL
LIN {X 0,Y 483.264,Z 465.813,A -85,B 0,C 180,E1 -6966.085,E2 -6966.085} C_VEL
LIN {X 0,Y 482.203,Z 459.366,A -85,B 0,C 180,E1 -6968.808,E2 -6968.808} C_VEL
LIN {X 0,Y 481.705,Z 456.485,A -85,B 0,C 180,E1 -6970.068,E2 -6970.068} C_VEL
LIN {X 0,Y 481.641,Z 456.491,A -85,B 0,C 180,E1 -6973.3,E2 -6973.3} C_VEL
LIN {X 0,Y 481.686,Z 456.484,A -85,B 0,C 180,E1 -6976.705,E2 -6976.705} C_VEL
LIN {X 0,Y 481.678,Z 456.484,A -85,B 0,C 180,E1 -6980.06,E2 -6980.06} C_VEL
LIN {X 0,Y 481.627,Z 456.491,A -85,B 0,C 180,E1 -6983.253,E2 -6983.253} C_VEL
LIN {X 0,Y 481.711,Z 456.481,A -85,B 0,C 180,E1 -6986.33,E2 -6986.33} C_VEL
LIN {X 0,Y 481.652,Z 456.487,A -85,B 0,C 180,E1 -6989.417,E2 -6989.417} C_VEL
LIN {X 0,Y 481.702,Z 456.483,A -85,B 0,C 180,E1 -6992.168,E2 -6992.168} C_VEL
LIN {X 0,Y 481.717,Z 456.481,A -85,B 0,C 180,E1 -6994.97,E2 -6994.97} C_VEL
LIN {X 0,Y 481.651,Z 456.489,A -85,B 0,C 180,E1 -6997.705,E2 -6997.705} C_VEL
LIN {X 0,Y 481.71,Z 456.481,A -85,B 0,C 180,E1 -7000.393,E2 -7000.393} C_VEL
LIN {X 0,Y 481.693,Z 456.483,A -85,B 0,C 180,E1 -7003.034,E2 -7003.034} C_VEL
LIN {X 0,Y 481.692,Z 456.484,A -85,B 0,C 180,E1 -7005.639,E2 -7005.639} C_VEL
LIN {X 0,Y 481.753,Z 456.475,A -85,B 0,C 180,E1 -7008.215,E2 -7008.215} C_VEL
LIN {X 0,Y 481.765,Z 456.474,A -85,B 0,C 180,E1 -7011.612,E2 -7011.612} C_VEL
LIN {X 0,Y 481.818,Z 456.468,A -85,B 0,C 180,E1 -7014.14,E2 -7014.14} C_VEL
LIN {X 0,Y 481.929,Z 456.452,A -85,B 0,C 180,E1 -7017.493,E2 -7017.493} C_VEL
LIN {X 0,Y 481.909,Z 456.457,A -85,B 0,C 180,E1 -7020.836,E2 -7020.836} C_VEL
LIN {X 0,Y 481.929,Z 456.455,A -85,B 0,C 180,E1 -7022.508,E2 -7022.508} C_VEL
LIN {X 0,Y 481.818,Z 456.468,A -85,B 0,C 180,E1 -7025.861,E2 -7025.861} C_VEL
LIN {X 0,Y 481.766,Z 456.474,A -85,B 0,C 180,E1 -7028.388,E2 -7028.388} C_VEL
LIN {X 0,Y 481.753,Z 456.474,A -85,B 0,C 180,E1 -7031.785,E2 -7031.785} C_VEL
LIN {X 0,Y 481.745,Z 456.478,A -85,B 0,C 180,E1 -7035.224,E2 -7035.224} C_VEL
LIN {X 0,Y 481.715,Z 456.481,A -85,B 0,C 180,E1 -7038.722,E2 -7038.722} C_VEL
LIN {X 0,Y 481.648,Z 456.49,A -85,B 0,C 180,E1 -7041.395,E2 -7041.395} C_VEL
LIN {X 0,Y 481.677,Z 456.485,A -85,B 0,C 180,E1 -7044.113,E2 -7044.113} C_VEL
LIN {X 0,Y 481.75,Z 456.475,A -85,B 0,C 180,E1 -7047.139,E2 -7047.139} C_VEL
LIN {X 0,Y 481.682,Z 456.486,A -85,B 0,C 180,E1 -7049.741,E2 -7049.741} C_VEL
LIN {X 0,Y 481.675,Z 456.487,A -85,B 0,C 180,E1 -7052.674,E2 -7052.674} C_VEL
LIN {X 0,Y 481.645,Z 456.491,A -85,B 0,C 180,E1 -7055.709,E2 -7055.709} C_VEL
LIN {X 0,Y 481.674,Z 456.487,A -85,B 0,C 180,E1 -7058.859,E2 -7058.859} C_VEL
LIN {X 0,Y 481.665,Z 456.489,A -85,B 0,C 180,E1 -7061.914,E2 -7061.914} C_VEL
LIN {X 0,Y 481.664,Z 456.487,A -85,B 0,C 180,E1 -7064.457,E2 -7064.457} C_VEL
LIN {X 0,Y 481.651,Z 456.489,A -85,B 0,C 180,E1 -7067.84,E2 -7067.84} C_VEL
LIN {X 0,Y 481.684,Z 456.485,A -85,B 0,C 180,E1 -7070.651,E2 -7070.651} C_VEL
LIN {X 0,Y 481.634,Z 456.49,A -85,B 0,C 180,E1 -7073.376,E2 -7073.376} C_VEL
LIN {X 0,Y 481.713,Z 456.481,A -85,B 0,C 180,E1 -7076.33,E2 -7076.33} C_VEL
LIN {X 0,Y 481.655,Z 456.489,A -85,B 0,C 180,E1 -7079.418,E2 -7079.418} C_VEL
LIN {X 0,Y 481.704,Z 456.486,A -85,B 0,C 180,E1 -7082.168,E2 -7082.168} C_VEL
LIN {X 0,Y 481.722,Z 456.481,A -85,B 0,C 180,E1 -7084.97,E2 -7084.97} C_VEL
LIN {X 0,Y 481.64,Z 456.488,A -85,B 0,C 180,E1 -7087.981,E2 -7087.981} C_VEL
LIN {X 0,Y 480.973,Z 456.573,A -85,B 0,C 180,E1 -7088.679,E2 -7088.679} C_VEL
LIN {X 0,Y 478.147,Z 456.926,A -85,B 0,C 180,E1 -7089.813,E2 -7089.813} C_VEL
LIN {X 0,Y 475.76,Z 457.223,A -85,B 0,C 180,E1 -7090.727,E2 -7090.727} C_VEL
LIN {X 0,Y 474.735,Z 457.351,A -85,B 0,C 180,E1 -7091.433,E2 -7091.433} C_VEL
LIN {X 0,Y 474.651,Z 457.361,A -85,B 0,C 180,E1 -7091.672,E2 -7091.672} C_VEL
LIN {X 0,Y 474.705,Z 457.356,A -85,B 0,C 180,E1 -7094.545,E2 -7094.545} C_VEL
LIN {X 0,Y 474.71,Z 457.355,A -85,B 0,C 180,E1 -7098.038,E2 -7098.038} C_VEL
LIN {X 0,Y 474.732,Z 457.35,A -85,B 0,C 180,E1 -7101.487,E2 -7101.487} C_VEL
LIN {X 0,Y 474.751,Z 457.347,A -85,B 0,C 180,E1 -7104.904,E2 -7104.904} C_VEL
LIN {X 0,Y 474.899,Z 457.332,A -85,B 0,C 180,E1 -7107.455,E2 -7107.455} C_VEL
LIN {X 0,Y 474.917,Z 457.329,A -85,B 0,C 180,E1 -7110,E2 -7110} C_VEL
LIN {X 0,Y 474.899,Z 457.329,A -85,B 0,C 180,E1 -7112.545,E2 -7112.545} C_VEL
LIN {X 0,Y 474.783,Z 457.344,A -85,B 0,C 180,E1 -7115.948,E2 -7115.948} C_VEL
LIN {X 0,Y 474.718,Z 457.351,A -85,B 0,C 180,E1 -7118.514,E2 -7118.514} C_VEL
LIN {X 0,Y 474.71,Z 457.353,A -85,B 0,C 180,E1 -7121.962,E2 -7121.962} C_VEL
LIN {X 0,Y 474.705,Z 457.353,A -85,B 0,C 180,E1 -7125.456,E2 -7125.456} C_VEL
LIN {X 0,Y 474.67,Z 457.359,A -85,B 0,C 180,E1 -7129.01,E2 -7129.01} C_VEL
LIN {X 0,Y 474.594,Z 457.368,A -85,B 0,C 180,E1 -7131.729,E2 -7131.729} C_VEL
LIN {X 0,Y 474.662,Z 457.358,A -85,B 0,C 180,E1 -7134.493,E2 -7134.493} C_VEL
LIN {X 0,Y 474.686,Z 457.356,A -85,B 0,C 180,E1 -7137.334,E2 -7137.334} C_VEL
LIN {X 0,Y 474.61,Z 457.365,A -85,B 0,C 180,E1 -7140.23,E2 -7140.23} C_VEL
LIN {X 0,Y 474.647,Z 457.363,A -85,B 0,C 180,E1 -7143.22,E2 -7143.22} C_VEL
LIN {X 0,Y 474.593,Z 457.368,A -85,B 0,C 180,E1 -7146.323,E2 -7146.323} C_VEL
LIN {X 0,Y 474.632,Z 457.364,A -85,B 0,C 180,E1 -7149.648,E2 -7149.648} C_VEL
LIN {X 0,Y 474.618,Z 457.364,A -85,B 0,C 180,E1 -7152.934,E2 -7152.934} C_VEL
LIN {X 0,Y 474.61,Z 457.366,A -85,B 0,C 180,E1 -7155.895,E2 -7155.895} C_VEL
LIN {X 0,Y 474.632,Z 457.364,A -85,B 0,C 180,E1 -7159.041,E2 -7159.041} C_VEL
LIN {X 0,Y 474.611,Z 457.369,A -85,B 0,C 180,E1 -7161.704,E2 -7161.704} C_VEL
LIN {X 0,Y 474.542,Z 457.375,A -85,B 0,C 180,E1 -7164.718,E2 -7164.718} C_VEL
LIN {X 0,Y 474.212,Z 457.419,A -85,B 0,C 180,E1 -7167.755,E2 -7167.755} C_VEL
LIN {X 0,Y 474.064,Z 457.578,A -85,B 0,C 180,E1 -7169.3,E2 -7169.3} C_VEL
LIN {X 0,Y 474.02,Z 461.074,A -85,B 0,C 180,E1 -7172.637,E2 -7172.637} C_VEL
LIN {X 0,Y 473.932,Z 464.078,A -85,B 0,C 180,E1 -7175.467,E2 -7175.467} C_VEL
LIN {X 0,Y 473.887,Z 467.069,A -85,B 0,C 180,E1 -7178.237,E2 -7178.237} C_VEL
LIN {X 0,Y 473.905,Z 470.781,A -85,B 0,C 180,E1 -7181.645,E2 -7181.645} C_VEL
LIN {X 0,Y 473.845,Z 474.501,A -85,B 0,C 180,E1 -7184.987,E2 -7184.987} C_VEL
LIN {X 0,Y 476.661,Z 487.642,A -85,B 0,C 180,E1 -7185.484,E2 -7185.484} C_VEL
LIN {X 0,Y 476.913,Z 492.995,A -85,B 0,C 180,E1 -7185.709,E2 -7185.709} C_VEL
LIN {X 0,Y 476.548,Z 505.808,A -85,B 0,C 180,E1 -7186.351,E2 -7186.351} C_VEL
LIN {X 0,Y 476.139,Z 517.228,A -85,B 0,C 180,E1 -7187.107,E2 -7187.107} C_VEL
LIN {X 0,Y 475.657,Z 528.656,A -85,B 0,C 180,E1 -7188.062,E2 -7188.062} C_VEL
LIN {X 0,Y 475.185,Z 538.91,A -85,B 0,C 180,E1 -7189.13,E2 -7189.13} C_VEL
LIN {X 0,Y 474.843,Z 547.25,A -85,B 0,C 180,E1 -7190.2,E2 -7190.2} C_VEL
LIN {X 0,Y 474.498,Z 555.419,A -85,B 0,C 180,E1 -7191.482,E2 -7191.482} C_VEL
LIN {X 0,Y 474.219,Z 561.996,A -85,B 0,C 180,E1 -7192.763,E2 -7192.763} C_VEL
LIN {X 0,Y 474.094,Z 567.225,A -85,B 0,C 180,E1 -7194.044,E2 -7194.044} C_VEL
LIN {X 0,Y 473.941,Z 571.29,A -85,B 0,C 180,E1 -7195.322,E2 -7195.322} C_VEL
LIN {X 0,Y 473.848,Z 574.301,A -85,B 0,C 180,E1 -7196.599,E2 -7196.599} C_VEL
LIN {X 0,Y 473.866,Z 575.754,A -85,B 0,C 180,E1 -7197.45,E2 -7197.45} C_VEL
LIN {X 0,Y 473.689,Z 577.452,A -85,B 0,C 180,E1 -7199.15,E2 -7199.15} C_VEL
LIN {X 0,Y 473.671,Z 577.718,A -85,B 0,C 180,E1 -7200,E2 -7200} C_VEL
LIN {X 0,Y 473.689,Z 577.548,A -85,B 0,C 180,E1 -7200.85,E2 -7200.85} C_VEL
LIN {X 0,Y 473.868,Z 576.016,A -85,B 0,C 180,E1 -7202.55,E2 -7202.55} C_VEL
LIN {X 0,Y 473.856,Z 574.663,A -85,B 0,C 180,E1 -7203.401,E2 -7203.401} C_VEL
LIN {X 0,Y 473.945,Z 571.791,A -85,B 0,C 180,E1 -7204.678,E2 -7204.678} C_VEL
LIN {X 0,Y 474.093,Z 567.878,A -85,B 0,C 180,E1 -7205.956,E2 -7205.956} C_VEL
LIN {X 0,Y 474.239,Z 562.813,A -85,B 0,C 180,E1 -7207.236,E2 -7207.236} C_VEL
LIN {X 0,Y 474.503,Z 556.405,A -85,B 0,C 180,E1 -7208.517,E2 -7208.517} C_VEL
LIN {X 0,Y 474.82,Z 548.416,A -85,B 0,C 180,E1 -7209.8,E2 -7209.8} C_VEL
LIN {X 0,Y 475.215,Z 540.25,A -85,B 0,C 180,E1 -7210.869,E2 -7210.869} C_VEL
LIN {X 0,Y 475.733,Z 530.26,A -85,B 0,C 180,E1 -7211.936,E2 -7211.936} C_VEL
LIN {X 0,Y 476.108,Z 520.386,A -85,B 0,C 180,E1 -7212.792,E2 -7212.792} C_VEL
LIN {X 0,Y 476.499,Z 509.63,A -85,B 0,C 180,E1 -7213.547,E2 -7213.547} C_VEL
LIN {X 0,Y 476.913,Z 497.054,A -85,B 0,C 180,E1 -7214.236,E2 -7214.236} C_VEL
LIN {X 0,Y 476.934,Z 489.136,A -85,B 0,C 180,E1 -7214.576,E2 -7214.576} C_VEL
LIN {X 0,Y 474.54,Z 478.38,A -85,B 0,C 180,E1 -7215.021,E2 -7215.021} C_VEL
LIN {X 0,Y 474.025,Z 476.186,A -85,B 0,C 180,E1 -7215.117,E2 -7215.117} C_VEL
LIN {X 0,Y 474.1,Z 473.008,A -85,B 0,C 180,E1 -7218.426,E2 -7218.426} C_VEL
LIN {X 0,Y 474.159,Z 470.644,A -85,B 0,C 180,E1 -7220.966,E2 -7220.966} C_VEL
LIN {X 0,Y 474.217,Z 468.314,A -85,B 0,C 180,E1 -7223.587,E2 -7223.587} C_VEL
LIN {X 0,Y 474.361,Z 465.964,A -85,B 0,C 180,E1 -7226.39,E2 -7226.39} C_VEL
LIN {X 0,Y 474.497,Z 463.711,A -85,B 0,C 180,E1 -7229.26,E2 -7229.26} C_VEL
LIN {X 0,Y 474.697,Z 461.45,A -85,B 0,C 180,E1 -7232.445,E2 -7232.445} C_VEL
LIN {X 0,Y 474.834,Z 459.642,A -85,B 0,C 180,E1 -7235.506,E2 -7235.506} C_VEL
LIN {X 0,Y 474.787,Z 458.44,A -85,B 0,C 180,E1 -7238.441,E2 -7238.441} C_VEL
LIN {X 0,Y 474.721,Z 457.931,A -85,B 0,C 180,E1 -7240.972,E2 -7240.972} C_VEL
LIN {X 0,Y 474.731,Z 458.111,A -85,B 0,C 180,E1 -7243.497,E2 -7243.497} C_VEL
LIN {X 0,Y 474.903,Z 459.055,A -85,B 0,C 180,E1 -7245.929,E2 -7245.929} C_VEL
LIN {X 0,Y 475.396,Z 461.426,A -85,B 0,C 180,E1 -7248.934,E2 -7248.934} C_VEL
LIN {X 0,Y 475.954,Z 464.759,A -85,B 0,C 180,E1 -7251.671,E2 -7251.671} C_VEL
LIN {X 0,Y 476.38,Z 468.92,A -85,B 0,C 180,E1 -7254.234,E2 -7254.234} C_VEL
LIN {X 0,Y 475.934,Z 474.29,A -85,B 0,C 180,E1 -7256.881,E2 -7256.881} C_VEL
LIN {X 0,Y 475.371,Z 481.083,A -85,B 0,C 180,E1 -7259.823,E2 -7259.823} C_VEL
LIN {X 0,Y 474.945,Z 489.648,A -85,B 0,C 180,E1 -7263.171,E2 -7263.171} C_VEL
LIN {X 0,Y 474.641,Z 497.343,A -85,B 0,C 180,E1 -7265.971,E2 -7265.971} C_VEL
LIN {X 0,Y 474.406,Z 506.589,A -85,B 0,C 180,E1 -7269.173,E2 -7269.173} C_VEL
LIN {X 0,Y 474.165,Z 515.977,A -85,B 0,C 180,E1 -7272.311,E2 -7272.311} C_VEL
LIN {X 0,Y 474.114,Z 523.769,A -85,B 0,C 180,E1 -7274.855,E2 -7274.855} C_VEL
LIN {X 0,Y 475.915,Z 538.152,A -85,B 0,C 180,E1 -7275.31,E2 -7275.31} C_VEL
LIN {X 0,Y 476.672,Z 544.893,A -85,B 0,C 180,E1 -7275.593,E2 -7275.593} C_VEL
LIN {X 0,Y 476.225,Z 558.097,A -85,B 0,C 180,E1 -7276.233,E2 -7276.233} C_VEL
LIN {X 0,Y 475.805,Z 569.868,A -85,B 0,C 180,E1 -7276.982,E2 -7276.982} C_VEL
LIN {X 0,Y 475.273,Z 581.883,A -85,B 0,C 180,E1 -7277.957,E2 -7277.957} C_VEL
LIN {X 0,Y 474.897,Z 591.378,A -85,B 0,C 180,E1 -7278.908,E2 -7278.908} C_VEL
LIN {X 0,Y 474.504,Z 600.202,A -85,B 0,C 180,E1 -7279.978,E2 -7279.978} C_VEL
LIN {X 0,Y 474.213,Z 608.784,A -85,B 0,C 180,E1 -7281.262,E2 -7281.262} C_VEL
LIN {X 0,Y 474.017,Z 615.706,A -85,B 0,C 180,E1 -7282.546,E2 -7282.546} C_VEL
LIN {X 0,Y 473.855,Z 622.062,A -85,B 0,C 180,E1 -7284.041,E2 -7284.041} C_VEL
LIN {X 0,Y 473.775,Z 626.187,A -85,B 0,C 180,E1 -7285.32,E2 -7285.32} C_VEL
LIN {X 0,Y 473.821,Z 629.245,A -85,B 0,C 180,E1 -7286.599,E2 -7286.599} C_VEL
LIN {X 0,Y 473.793,Z 630.702,A -85,B 0,C 180,E1 -7287.449,E2 -7287.449} C_VEL
LIN {X 0,Y 473.758,Z 631.748,A -85,B 0,C 180,E1 -7288.3,E2 -7288.3} C_VEL
LIN {X 0,Y 473.688,Z 632.394,A -85,B 0,C 180,E1 -7289.15,E2 -7289.15} C_VEL
LIN {X 0,Y 473.669,Z 632.636,A -85,B 0,C 180,E1 -7290,E2 -7290} C_VEL
LIN {X 0,Y 473.758,Z 631.834,A -85,B 0,C 180,E1 -7291.7,E2 -7291.7} C_VEL
LIN {X 0,Y 473.783,Z 630.835,A -85,B 0,C 180,E1 -7292.55,E2 -7292.55} C_VEL
LIN {X 0,Y 473.82,Z 629.418,A -85,B 0,C 180,E1 -7293.401,E2 -7293.401} C_VEL
LIN {X 0,Y 473.774,Z 626.434,A -85,B 0,C 180,E1 -7294.68,E2 -7294.68} C_VEL
LIN {X 0,Y 473.854,Z 622.392,A -85,B 0,C 180,E1 -7295.959,E2 -7295.959} C_VEL
LIN {X 0,Y 474.017,Z 616.158,A -85,B 0,C 180,E1 -7297.454,E2 -7297.454} C_VEL
LIN {X 0,Y 474.243,Z 609.361,A -85,B 0,C 180,E1 -7298.737,E2 -7298.737} C_VEL
LIN {X 0,Y 474.522,Z 600.924,A -85,B 0,C 180,E1 -7300.022,E2 -7300.022} C_VEL
LIN {X 0,Y 474.934,Z 592.245,A -85,B 0,C 180,E1 -7301.091,E2 -7301.091} C_VEL
LIN {X 0,Y 475.351,Z 581.815,A -85,B 0,C 180,E1 -7302.142,E2 -7302.142} C_VEL
LIN {X 0,Y 475.827,Z 571.354,A -85,B 0,C 180,E1 -7302.995,E2 -7302.995} C_VEL
LIN {X 0,Y 476.301,Z 559.452,A -85,B 0,C 180,E1 -7303.764,E2 -7303.764} C_VEL
LIN {X 0,Y 476.789,Z 546.33,A -85,B 0,C 180,E1 -7304.403,E2 -7304.403} C_VEL
LIN {X 0,Y 476.331,Z 540.718,A -85,B 0,C 180,E1 -7304.636,E2 -7304.636} C_VEL
LIN {X 0,Y 474.476,Z 527.611,A -85,B 0,C 180,E1 -7305.078,E2 -7305.078} C_VEL
LIN {X 0,Y 474.167,Z 525.157,A -85,B 0,C 180,E1 -7305.143,E2 -7305.143} C_VEL
LIN {X 0,Y 474.341,Z 515.184,A -85,B 0,C 180,E1 -7308.513,E2 -7308.513} C_VEL
LIN {X 0,Y 474.603,Z 505.842,A -85,B 0,C 180,E1 -7311.728,E2 -7311.728} C_VEL
LIN {X 0,Y 474.923,Z 496.712,A -85,B 0,C 180,E1 -7314.945,E2 -7314.945} C_VEL
LIN {X 0,Y 475.339,Z 487.595,A -85,B 0,C 180,E1 -7318.238,E2 -7318.238} C_VEL
LIN {X 0,Y 475.74,Z 479.838,A -85,B 0,C 180,E1 -7321.134,E2 -7321.134} C_VEL
LIN {X 0,Y 476.139,Z 472.09,A -85,B 0,C 180,E1 -7324.118,E2 -7324.118} C_VEL
LIN {X 0,Y 476.264,Z 466.927,A -85,B 0,C 180,E1 -7326.176,E2 -7326.176} C_VEL
LIN {X 0,Y 475.197,Z 460.471,A -85,B 0,C 180,E1 -7328.944,E2 -7328.944} C_VEL
LIN {X 0,Y 474.651,Z 457.363,A -85,B 0,C 180,E1 -7330.394,E2 -7330.394} C_VEL
LIN {X 0,Y 474.603,Z 457.367,A -85,B 0,C 180,E1 -7333.481,E2 -7333.481} C_VEL
LIN {X 0,Y 474.637,Z 457.363,A -85,B 0,C 180,E1 -7336.514,E2 -7336.514} C_VEL
LIN {X 0,Y 474.621,Z 457.365,A -85,B 0,C 180,E1 -7339.343,E2 -7339.343} C_VEL
LIN {X 0,Y 474.591,Z 457.37,A -85,B 0,C 180,E1 -7342.616,E2 -7342.616} C_VEL
LIN {X 0,Y 474.633,Z 457.363,A -85,B 0,C 180,E1 -7345.759,E2 -7345.759} C_VEL
LIN {X 0,Y 474.6,Z 457.369,A -85,B 0,C 180,E1 -7348.782,E2 -7348.782} C_VEL
LIN {X 0,Y 474.648,Z 457.362,A -85,B 0,C 180,E1 -7351.718,E2 -7351.718} C_VEL
LIN {X 0,Y 474.671,Z 457.36,A -85,B 0,C 180,E1 -7354.578,E2 -7354.578} C_VEL
LIN {X 0,Y 474.602,Z 457.366,A -85,B 0,C 180,E1 -7357.355,E2 -7357.355} C_VEL
LIN {X 0,Y 474.659,Z 457.36,A -85,B 0,C 180,E1 -7360.09,E2 -7360.09} C_VEL
LIN {X 0,Y 474.653,Z 457.362,A -85,B 0,C 180,E1 -7362.775,E2 -7362.775} C_VEL
LIN {X 0,Y 474.651,Z 457.362,A -85,B 0,C 180,E1 -7365.421,E2 -7365.421} C_VEL
LIN {X 0,Y 474.706,Z 457.353,A -85,B 0,C 180,E1 -7368.038,E2 -7368.038} C_VEL
LIN {X 0,Y 474.73,Z 457.35,A -85,B 0,C 180,E1 -7371.487,E2 -7371.487} C_VEL
LIN {X 0,Y 474.781,Z 457.345,A -85,B 0,C 180,E1 -7374.053,E2 -7374.053} C_VEL
LIN {X 0,Y 474.896,Z 457.328,A -85,B 0,C 180,E1 -7377.456,E2 -7377.456} C_VEL
LIN {X 0,Y 474.915,Z 457.33,A -85,B 0,C 180,E1 -7380,E2 -7380} C_VEL
LIN {X 0,Y 474.896,Z 457.331,A -85,B 0,C 180,E1 -7382.545,E2 -7382.545} C_VEL
LIN {X 0,Y 474.781,Z 457.345,A -85,B 0,C 180,E1 -7385.948,E2 -7385.948} C_VEL
LIN {X 0,Y 474.731,Z 457.351,A -85,B 0,C 180,E1 -7388.514,E2 -7388.514} C_VEL
LIN {X 0,Y 474.707,Z 457.353,A -85,B 0,C 180,E1 -7391.963,E2 -7391.963} C_VEL
LIN {X 0,Y 474.703,Z 457.355,A -85,B 0,C 180,E1 -7395.456,E2 -7395.456} C_VEL
LIN {X 0,Y 474.668,Z 457.357,A -85,B 0,C 180,E1 -7399.01,E2 -7399.01} C_VEL
LIN {X 0,Y 474.592,Z 457.37,A -85,B 0,C 180,E1 -7401.729,E2 -7401.729} C_VEL
LIN {X 0,Y 474.66,Z 457.362,A -85,B 0,C 180,E1 -7404.493,E2 -7404.493} C_VEL
LIN {X 0,Y 474.702,Z 457.353,A -85,B 0,C 180,E1 -7407.339,E2 -7407.339} C_VEL
LIN {X 0,Y 474.608,Z 457.368,A -85,B 0,C 180,E1 -7410.81,E2 -7410.81} C_VEL
LIN {X 0,Y 474.641,Z 457.363,A -85,B 0,C 180,E1 -7413.984,E2 -7413.984} C_VEL
LIN {X 0,Y 474.578,Z 457.372,A -85,B 0,C 180,E1 -7416.9,E2 -7416.9} C_VEL
LIN {X 0,Y 474.621,Z 457.363,A -85,B 0,C 180,E1 -7419.646,E2 -7419.646} C_VEL
LIN {X 0,Y 474.639,Z 457.362,A -85,B 0,C 180,E1 -7422.932,E2 -7422.932} C_VEL
LIN {X 0,Y 474.613,Z 457.365,A -85,B 0,C 180,E1 -7425.895,E2 -7425.895} C_VEL
LIN {X 0,Y 474.631,Z 457.362,A -85,B 0,C 180,E1 -7429.041,E2 -7429.041} C_VEL
LIN {X 0,Y 474.614,Z 457.366,A -85,B 0,C 180,E1 -7431.704,E2 -7431.704} C_VEL
LIN {X 0,Y 474.633,Z 457.362,A -85,B 0,C 180,E1 -7434.726,E2 -7434.726} C_VEL
LIN {X 0,Y 474.639,Z 457.364,A -85,B 0,C 180,E1 -7437.788,E2 -7437.788} C_VEL
LIN {X 0,Y 474.628,Z 457.363,A -85,B 0,C 180,E1 -7440.885,E2 -7440.885} C_VEL
LIN {X 0,Y 474.665,Z 457.36,A -85,B 0,C 180,E1 -7443.629,E2 -7443.629} C_VEL
LIN {X 0,Y 474.64,Z 457.364,A -85,B 0,C 180,E1 -7446.642,E2 -7446.642} C_VEL
LIN {X 0,Y 474.659,Z 457.362,A -85,B 0,C 180,E1 -7450.09,E2 -7450.09} C_VEL
LIN {X 0,Y 474.651,Z 457.361,A -85,B 0,C 180,E1 -7451.672,E2 -7451.672} C_VEL
LIN {X 0,Y 473.984,Z 457.446,A -85,B 0,C 180,E1 -7452.381,E2 -7452.381} C_VEL
LIN {X 0,Y 471.137,Z 457.8,A -85,B 0,C 180,E1 -7453.533,E2 -7453.533} C_VEL
LIN {X 0,Y 468.727,Z 458.102,A -85,B 0,C 180,E1 -7454.461,E2 -7454.461} C_VEL
LIN {X 0,Y 467.688,Z 458.227,A -85,B 0,C 180,E1 -7455.178,E2 -7455.178} C_VEL
LIN {X 0,Y 467.602,Z 458.238,A -85,B 0,C 180,E1 -7455.421,E2 -7455.421} C_VEL
LIN {X 0,Y 467.657,Z 458.232,A -85,B 0,C 180,E1 -7458.734,E2 -7458.734} C_VEL
LIN {X 0,Y 467.685,Z 458.229,A -85,B 0,C 180,E1 -7461.357,E2 -7461.357} C_VEL
LIN {X 0,Y 467.726,Z 458.226,A -85,B 0,C 180,E1 -7463.962,E2 -7463.962} C_VEL
LIN {X 0,Y 467.864,Z 458.208,A -85,B 0,C 180,E1 -7467.417,E2 -7467.417} C_VEL
LIN {X 0,Y 467.888,Z 458.205,A -85,B 0,C 180,E1 -7470,E2 -7470} C_VEL
LIN {X 0,Y 467.864,Z 458.205,A -85,B 0,C 180,E1 -7472.583,E2 -7472.583} C_VEL
LIN {X 0,Y 467.747,Z 458.221,A -85,B 0,C 180,E1 -7476.037,E2 -7476.037} C_VEL
LIN {X 0,Y 467.676,Z 458.228,A -85,B 0,C 180,E1 -7478.643,E2 -7478.643} C_VEL
LIN {X 0,Y 467.661,Z 458.232,A -85,B 0,C 180,E1 -7482.145,E2 -7482.145} C_VEL
LIN {X 0,Y 467.644,Z 458.235,A -85,B 0,C 180,E1 -7485.695,E2 -7485.695} C_VEL
LIN {X 0,Y 467.622,Z 458.237,A -85,B 0,C 180,E1 -7488.765,E2 -7488.765} C_VEL
LIN {X 0,Y 467.585,Z 458.24,A -85,B 0,C 180,E1 -7491.268,E2 -7491.268} C_VEL
LIN {X 0,Y 467.577,Z 458.243,A -85,B 0,C 180,E1 -7493.943,E2 -7493.943} C_VEL
LIN {X 0,Y 467.621,Z 458.237,A -85,B 0,C 180,E1 -7496.8,E2 -7496.8} C_VEL
LIN {X 0,Y 467.559,Z 458.246,A -85,B 0,C 180,E1 -7499.738,E2 -7499.738} C_VEL
LIN {X 0,Y 467.588,Z 458.241,A -85,B 0,C 180,E1 -7502.758,E2 -7502.758} C_VEL
LIN {X 0,Y 467.558,Z 458.246,A -85,B 0,C 180,E1 -7505.89,E2 -7505.89} C_VEL
LIN {X 0,Y 467.587,Z 458.241,A -85,B 0,C 180,E1 -7509.145,E2 -7509.145} C_VEL
LIN {X 0,Y 467.591,Z 458.24,A -85,B 0,C 180,E1 -7512.567,E2 -7512.567} C_VEL
LIN {X 0,Y 467.57,Z 458.241,A -85,B 0,C 180,E1 -7515.052,E2 -7515.052} C_VEL
LIN {X 0,Y 467.593,Z 458.241,A -85,B 0,C 180,E1 -7517.44,E2 -7517.44} C_VEL
LIN {X 0,Y 467.585,Z 458.239,A -85,B 0,C 180,E1 -7520.855,E2 -7520.855} C_VEL
LIN {X 0,Y 467.502,Z 458.251,A -85,B 0,C 180,E1 -7524.105,E2 -7524.105} C_VEL
LIN {X 0,Y 467.333,Z 458.275,A -85,B 0,C 180,E1 -7526.191,E2 -7526.191} C_VEL
LIN {X 0,Y 467.029,Z 458.314,A -85,B 0,C 180,E1 -7529.226,E2 -7529.226} C_VEL
LIN {X 0,Y 466.972,Z 461.69,A -85,B 0,C 180,E1 -7532.618,E2 -7532.618} C_VEL
LIN {X 0,Y 466.875,Z 464.27,A -85,B 0,C 180,E1 -7535.071,E2 -7535.071} C_VEL
LIN {X 0,Y 466.824,Z 467.297,A -85,B 0,C 180,E1 -7537.89,E2 -7537.89} C_VEL
LIN {X 0,Y 466.79,Z 470.282,A -85,B 0,C 180,E1 -7540.656,E2 -7540.656} C_VEL
LIN {X 0,Y 466.746,Z 473.293,A -85,B 0,C 180,E1 -7543.376,E2 -7543.376} C_VEL
LIN {X 0,Y 466.792,Z 474.891,A -85,B 0,C 180,E1 -7544.77,E2 -7544.77} C_VEL
LIN {X 0,Y 469.773,Z 488.684,A -85,B 0,C 180,E1 -7545.308,E2 -7545.308} C_VEL
LIN {X 0,Y 470.003,Z 494.244,A -85,B 0,C 180,E1 -7545.55,E2 -7545.55} C_VEL
LIN {X 0,Y 469.643,Z 505.863,A -85,B 0,C 180,E1 -7546.147,E2 -7546.147} C_VEL
LIN {X 0,Y 469.211,Z 517.156,A -85,B 0,C 180,E1 -7546.898,E2 -7546.898} C_VEL
LIN {X 0,Y 468.732,Z 528.822,A -85,B 0,C 180,E1 -7547.883,E2 -7547.883} C_VEL
LIN {X 0,Y 468.215,Z 539.13,A -85,B 0,C 180,E1 -7548.966,E2 -7548.966} C_VEL
LIN {X 0,Y 467.853,Z 547.504,A -85,B 0,C 180,E1 -7550.052,E2 -7550.052} C_VEL
LIN {X 0,Y 467.474,Z 555.705,A -85,B 0,C 180,E1 -7551.353,E2 -7551.353} C_VEL
LIN {X 0,Y 467.175,Z 562.311,A -85,B 0,C 180,E1 -7552.653,E2 -7552.653} C_VEL
LIN {X 0,Y 467.049,Z 567.566,A -85,B 0,C 180,E1 -7553.953,E2 -7553.953} C_VEL
LIN {X 0,Y 466.862,Z 571.654,A -85,B 0,C 180,E1 -7555.251,E2 -7555.251} C_VEL
LIN {X 0,Y 466.786,Z 574.68,A -85,B 0,C 180,E1 -7556.547,E2 -7556.547} C_VEL
LIN {X 0,Y 466.79,Z 576.147,A -85,B 0,C 180,E1 -7557.411,E2 -7557.411} C_VEL
LIN {X 0,Y 466.621,Z 577.858,A -85,B 0,C 180,E1 -7559.137,E2 -7559.137} C_VEL
LIN {X 0,Y 466.6,Z 578.132,A -85,B 0,C 180,E1 -7560,E2 -7560} C_VEL
LIN {X 0,Y 466.62,Z 577.968,A -85,B 0,C 180,E1 -7560.863,E2 -7560.863} C_VEL
LIN {X 0,Y 466.809,Z 576.442,A -85,B 0,C 180,E1 -7562.589,E2 -7562.589} C_VEL
LIN {X 0,Y 466.794,Z 575.093,A -85,B 0,C 180,E1 -7563.453,E2 -7563.453} C_VEL
LIN {X 0,Y 466.885,Z 572.221,A -85,B 0,C 180,E1 -7564.749,E2 -7564.749} C_VEL
LIN {X 0,Y 467.049,Z 568.304,A -85,B 0,C 180,E1 -7566.046,E2 -7566.046} C_VEL
LIN {X 0,Y 467.212,Z 563.232,A -85,B 0,C 180,E1 -7567.346,E2 -7567.346} C_VEL
LIN {X 0,Y 467.509,Z 556.812,A -85,B 0,C 180,E1 -7568.646,E2 -7568.646} C_VEL
LIN {X 0,Y 467.85,Z 548.811,A -85,B 0,C 180,E1 -7569.948,E2 -7569.948} C_VEL
LIN {X 0,Y 468.256,Z 540.634,A -85,B 0,C 180,E1 -7571.032,E2 -7571.032} C_VEL
LIN {X 0,Y 468.814,Z 530.649,A -85,B 0,C 180,E1 -7572.115,E2 -7572.115} C_VEL
LIN {X 0,Y 469.237,Z 519.162,A -85,B 0,C 180,E1 -7573.116,E2 -7573.116} C_VEL
LIN {X 0,Y 469.671,Z 508.554,A -85,B 0,C 180,E1 -7573.852,E2 -7573.852} C_VEL
LIN {X 0,Y 470.112,Z 496.541,A -85,B 0,C 180,E1 -7574.501,E2 -7574.501} C_VEL
LIN {X 0,Y 470.119,Z 490.443,A -85,B 0,C 180,E1 -7574.77,E2 -7574.77} C_VEL
LIN {X 0,Y 467.925,Z 480.503,A -85,B 0,C 180,E1 -7575.206,E2 -7575.206} C_VEL
LIN {X 0,Y 466.98,Z 476.735,A -85,B 0,C 180,E1 -7575.37,E2 -7575.37} C_VEL
LIN {X 0,Y 467.04,Z 473.718,A -85,B 0,C 180,E1 -7578.554,E2 -7578.554} C_VEL
LIN {X 0,Y 467.114,Z 471.34,A -85,B 0,C 180,E1 -7581.167,E2 -7581.167} C_VEL
LIN {X 0,Y 467.19,Z 468.931,A -85,B 0,C 180,E1 -7583.964,E2 -7583.964} C_VEL
LIN {X 0,Y 467.352,Z 466.612,A -85,B 0,C 180,E1 -7586.817,E2 -7586.817} C_VEL
LIN {X 0,Y 467.508,Z 464.414,A -85,B 0,C 180,E1 -7589.741,E2 -7589.741} C_VEL
LIN {X 0,Y 467.727,Z 462.408,A -85,B 0,C 180,E1 -7592.747,E2 -7592.747} C_VEL
LIN {X 0,Y 467.809,Z 461.228,A -85,B 0,C 180,E1 -7594.812,E2 -7594.812} C_VEL
LIN {X 0,Y 467.829,Z 459.904,A -85,B 0,C 180,E1 -7598.019,E2 -7598.019} C_VEL
LIN {X 0,Y 467.776,Z 459.357,A -85,B 0,C 180,E1 -7601.304,E2 -7601.304} C_VEL
LIN {X 0,Y 467.838,Z 459.741,A -85,B 0,C 180,E1 -7603.857,E2 -7603.857} C_VEL
LIN {X 0,Y 468.026,Z 460.845,A -85,B 0,C 180,E1 -7606.31,E2 -7606.31} C_VEL
LIN {X 0,Y 468.416,Z 462.74,A -85,B 0,C 180,E1 -7608.687,E2 -7608.687} C_VEL
LIN {X 0,Y 468.902,Z 465.659,A -85,B 0,C 180,E1 -7611.205,E2 -7611.205} C_VEL
LIN {X 0,Y 469.284,Z 468.628,A -85,B 0,C 180,E1 -7613.199,E2 -7613.199} C_VEL
